ABB RAPID module: P902.mod

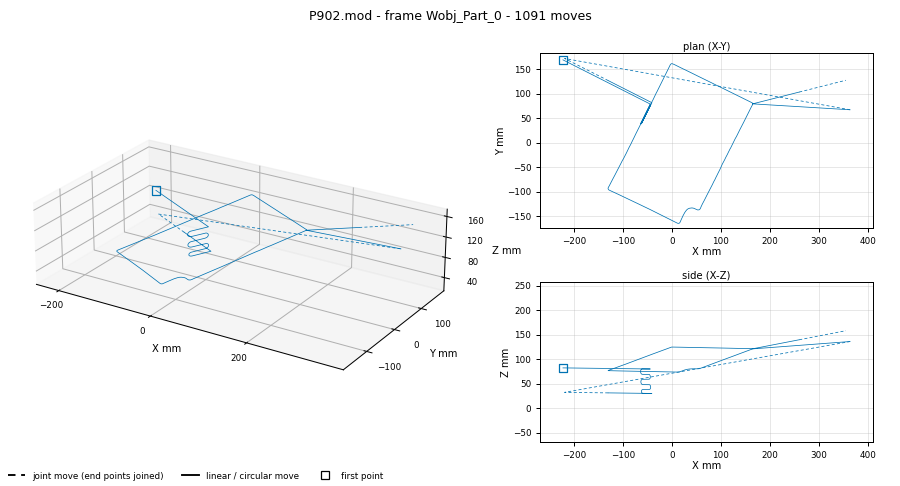
[picture p0: tool path of P902.mod in frame Wobj_Part_0, 1091 of 1101 moves have a stored position in this frame; points joined in program order, loops and branches not executed]
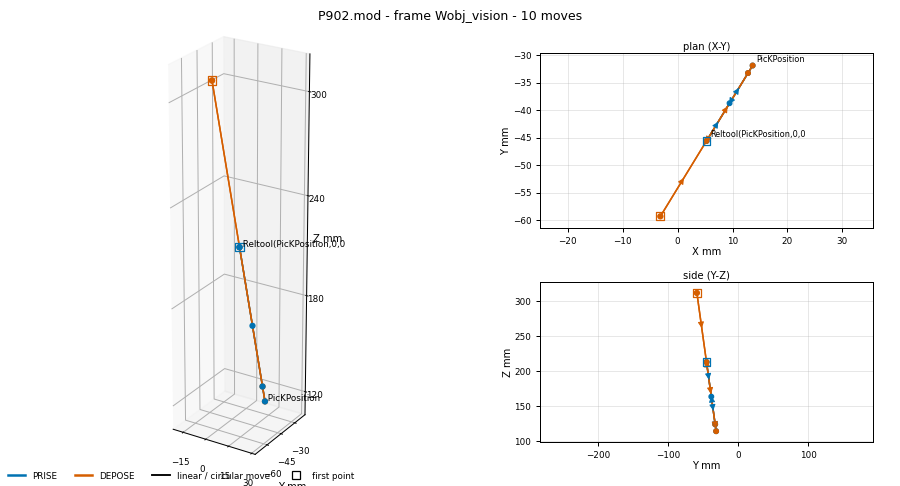
[picture p1: tool path of P902.mod in frame Wobj_vision, 10 of 1101 moves have a stored position in this frame; points joined in program order, loops and branches not executed]
MODULE P902

    ! Nom         :P902
    ! Description :
    ! Créé le     :01/06/2023 14:34:15

    LOCAL CONST SPEEDDATA VitesseLente :=[10,500,0,0];
	LOCAL CONST SPEEDDATA VitesseRapide :=[30,500,0,0];
	LOCAL CONST SPEEDDATA VitesseTronconnage :=[2,500,0,0];
	LOCAL CONST SPEEDDATA VitesseTronconnageApp :=[10,500,0,0];
    !
    !Point de prise
    LOCAL PERS Robtarget PicKPosition := [[13.6622090132406,-31.8672401655374,114.53373902136],[0.0717783424878255,-0.517500201429471,0.851863865981831,0.037004930815311],[0,0,0,0],[8.999999E+09,8.999999E+09,8.999999E+09,8.999999E+09,8.999999E+09,8.999999E+09]];
	LOCAL PERS Pose Ref := [[0,0,0],[1,0,0,0]];
    !
    !Declaration des points de meulage

    !Tr_meulage_motif_1 : Meulage d'un motif
    LOCAL CONST Robtarget Tr_meulage_motif_1_0 := [[-44.4600078125,78.776296875,79.8267421875],[0.368121083594183,-0.372259670766582,0.605815460428718,-0.599080322861418],[0,0,0,0],[8.999999E+09,8.999999E+09,8.999999E+09,8.999999E+09,8.999999E+09,8.999999E+09]];
    LOCAL CONST Robtarget Tr_meulage_motif_1_1 := [[-44.90398828125,77.8802578125,79.82678125],[0.368121083594183,-0.372259670766582,0.605815460428718,-0.599080322861418],[0,0,0,0],[8.999999E+09,8.999999E+09,8.999999E+09,8.999999E+09,8.999999E+09,8.999999E+09]];
    LOCAL CONST Robtarget Tr_meulage_motif_1_2 := [[-45.34796484375,76.98421875,79.8268203125],[0.368121083594183,-0.372259670766582,0.605815460428718,-0.599080322861418],[0,0,0,0],[8.999999E+09,8.999999E+09,8.999999E+09,8.999999E+09,8.999999E+09,8.999999E+09]];
    LOCAL CONST Robtarget Tr_meulage_motif_1_3 := [[-45.7919453125,76.0881796875,79.8268515625],[0.368121083594183,-0.372259670766582,0.605815460428718,-0.599080322861418],[0,0,0,0],[8.999999E+09,8.999999E+09,8.999999E+09,8.999999E+09,8.999999E+09,8.999999E+09]];
    LOCAL CONST Robtarget Tr_meulage_motif_1_4 := [[-46.23592578125,75.1921484375,79.826890625],[0.368121083594183,-0.372259670766582,0.605815460428718,-0.599080322861418],[0,0,0,0],[8.999999E+09,8.999999E+09,8.999999E+09,8.999999E+09,8.999999E+09,8.999999E+09]];
    LOCAL CONST Robtarget Tr_meulage_motif_1_5 := [[-46.67990234375,74.296109375,79.8269296875],[0.368121083594183,-0.372259670766582,0.605815460428718,-0.599080322861418],[0,0,0,0],[8.999999E+09,8.999999E+09,8.999999E+09,8.999999E+09,8.999999E+09,8.999999E+09]];
    LOCAL CONST Robtarget Tr_meulage_motif_1_6 := [[-47.1238828125,73.4000703125,79.82696875],[0.368121083594183,-0.372259670766582,0.605815460428718,-0.599080322861418],[0,0,0,0],[8.999999E+09,8.999999E+09,8.999999E+09,8.999999E+09,8.999999E+09,8.999999E+09]];
    LOCAL CONST Robtarget Tr_meulage_motif_1_7 := [[-47.567859375,72.50403125,79.827],[0.368121083594183,-0.372259670766582,0.605815460428718,-0.599080322861418],[0,0,0,0],[8.999999E+09,8.999999E+09,8.999999E+09,8.999999E+09,8.999999E+09,8.999999E+09]];
    LOCAL CONST Robtarget Tr_meulage_motif_1_8 := [[-48.01183984375,71.608,79.8270390625],[0.368121083594183,-0.372259670766582,0.605815460428718,-0.599080322861418],[0,0,0,0],[8.999999E+09,8.999999E+09,8.999999E+09,8.999999E+09,8.999999E+09,8.999999E+09]];
    LOCAL CONST Robtarget Tr_meulage_motif_1_9 := [[-48.4558203125,70.7119609375,79.827078125],[0.368121083594183,-0.372259670766582,0.605815460428718,-0.599080322861418],[0,0,0,0],[8.999999E+09,8.999999E+09,8.999999E+09,8.999999E+09,8.999999E+09,8.999999E+09]];
    LOCAL CONST Robtarget Tr_meulage_motif_1_10 := [[-48.899796875,69.815921875,79.8271171875],[0.368121083594183,-0.372259670766582,0.605815460428718,-0.599080322861418],[0,0,0,0],[8.999999E+09,8.999999E+09,8.999999E+09,8.999999E+09,8.999999E+09,8.999999E+09]];
    LOCAL CONST Robtarget Tr_meulage_motif_1_11 := [[-49.34377734375,68.9198828125,79.8271484375],[0.368121083594183,-0.372259670766582,0.605815460428718,-0.599080322861418],[0,0,0,0],[8.999999E+09,8.999999E+09,8.999999E+09,8.999999E+09,8.999999E+09,8.999999E+09]];
    LOCAL CONST Robtarget Tr_meulage_motif_1_12 := [[-49.78775390625,68.02384375,79.8271875],[0.368121083594183,-0.372259670766582,0.605815460428718,-0.599080322861418],[0,0,0,0],[8.999999E+09,8.999999E+09,8.999999E+09,8.999999E+09,8.999999E+09,8.999999E+09]];
    LOCAL CONST Robtarget Tr_meulage_motif_1_13 := [[-50.231734375,67.1278125,79.8272265625],[0.368121083594183,-0.372259670766582,0.605815460428718,-0.599080322861418],[0,0,0,0],[8.999999E+09,8.999999E+09,8.999999E+09,8.999999E+09,8.999999E+09,8.999999E+09]];
    LOCAL CONST Robtarget Tr_meulage_motif_1_14 := [[-50.67571484375,66.2317734375,79.827265625],[0.368121083594183,-0.372259670766582,0.605815460428718,-0.599080322861418],[0,0,0,0],[8.999999E+09,8.999999E+09,8.999999E+09,8.999999E+09,8.999999E+09,8.999999E+09]];
    LOCAL CONST Robtarget Tr_meulage_motif_1_15 := [[-51.11969140625,65.335734375,79.827296875],[0.368121083594183,-0.372259670766582,0.605815460428718,-0.599080322861418],[0,0,0,0],[8.999999E+09,8.999999E+09,8.999999E+09,8.999999E+09,8.999999E+09,8.999999E+09]];
    LOCAL CONST Robtarget Tr_meulage_motif_1_16 := [[-51.563671875,64.43969921875,79.8273359375],[0.368121083594183,-0.372259670766582,0.605815460428718,-0.599080322861418],[0,0,0,0],[8.999999E+09,8.999999E+09,8.999999E+09,8.999999E+09,8.999999E+09,8.999999E+09]];
    LOCAL CONST Robtarget Tr_meulage_motif_1_17 := [[-52.00765234375,63.54366015625,79.827375],[0.368121083594183,-0.372259670766582,0.605815460428718,-0.599080322861418],[0,0,0,0],[8.999999E+09,8.999999E+09,8.999999E+09,8.999999E+09,8.999999E+09,8.999999E+09]];
    LOCAL CONST Robtarget Tr_meulage_motif_1_18 := [[-52.45162890625,62.647625,79.8274140625],[0.368121083594183,-0.372259670766582,0.605815460428718,-0.599080322861418],[0,0,0,0],[8.999999E+09,8.999999E+09,8.999999E+09,8.999999E+09,8.999999E+09,8.999999E+09]];
    LOCAL CONST Robtarget Tr_meulage_motif_1_19 := [[-52.895609375,61.7515859375,79.8274453125],[0.368121083594183,-0.372259670766582,0.605815460428718,-0.599080322861418],[0,0,0,0],[8.999999E+09,8.999999E+09,8.999999E+09,8.999999E+09,8.999999E+09,8.999999E+09]];
    LOCAL CONST Robtarget Tr_meulage_motif_1_20 := [[-53.3395859375,60.85555078125,79.827484375],[0.368121083594183,-0.372259670766582,0.605815460428718,-0.599080322861418],[0,0,0,0],[8.999999E+09,8.999999E+09,8.999999E+09,8.999999E+09,8.999999E+09,8.999999E+09]];
    LOCAL CONST Robtarget Tr_meulage_motif_1_21 := [[-53.78356640625,59.95951171875,79.8275234375],[0.368121083594183,-0.372259670766582,0.605815460428718,-0.599080322861418],[0,0,0,0],[8.999999E+09,8.999999E+09,8.999999E+09,8.999999E+09,8.999999E+09,8.999999E+09]];
    LOCAL CONST Robtarget Tr_meulage_motif_1_22 := [[-54.227546875,59.0634765625,79.8275625],[0.368121083594183,-0.372259670766582,0.605815460428718,-0.599080322861418],[0,0,0,0],[8.999999E+09,8.999999E+09,8.999999E+09,8.999999E+09,8.999999E+09,8.999999E+09]];
    LOCAL CONST Robtarget Tr_meulage_motif_1_23 := [[-54.6715234375,58.1674375,79.82759375],[0.368121083594183,-0.372259670766582,0.605815460428718,-0.599080322861418],[0,0,0,0],[8.999999E+09,8.999999E+09,8.999999E+09,8.999999E+09,8.999999E+09,8.999999E+09]];
    LOCAL CONST Robtarget Tr_meulage_motif_1_24 := [[-55.11550390625,57.27140234375,79.8276328125],[0.368121083594183,-0.372259670766582,0.605815460428718,-0.599080322861418],[0,0,0,0],[8.999999E+09,8.999999E+09,8.999999E+09,8.999999E+09,8.999999E+09,8.999999E+09]];
    LOCAL CONST Robtarget Tr_meulage_motif_1_25 := [[-55.55948046875,56.37536328125,79.827671875],[0.368121083594183,-0.372259670766582,0.605815460428718,-0.599080322861418],[0,0,0,0],[8.999999E+09,8.999999E+09,8.999999E+09,8.999999E+09,8.999999E+09,8.999999E+09]];
    LOCAL CONST Robtarget Tr_meulage_motif_1_26 := [[-56.0034609375,55.479328125,79.8277109375],[0.368121083594183,-0.372259670766582,0.605815460428718,-0.599080322861418],[0,0,0,0],[8.999999E+09,8.999999E+09,8.999999E+09,8.999999E+09,8.999999E+09,8.999999E+09]];
    LOCAL CONST Robtarget Tr_meulage_motif_1_27 := [[-56.44744140625,54.5832890625,79.82775],[0.368121083594183,-0.372259670766582,0.605815460428718,-0.599080322861418],[0,0,0,0],[8.999999E+09,8.999999E+09,8.999999E+09,8.999999E+09,8.999999E+09,8.999999E+09]];
    LOCAL CONST Robtarget Tr_meulage_motif_1_28 := [[-56.89141796875,53.68725390625,79.82778125],[0.368121083594183,-0.372259670766582,0.605815460428718,-0.599080322861418],[0,0,0,0],[8.999999E+09,8.999999E+09,8.999999E+09,8.999999E+09,8.999999E+09,8.999999E+09]];
    LOCAL CONST Robtarget Tr_meulage_motif_1_29 := [[-57.3353984375,52.79121484375,79.8278203125],[0.368121083594183,-0.372259670766582,0.605815460428718,-0.599080322861418],[0,0,0,0],[8.999999E+09,8.999999E+09,8.999999E+09,8.999999E+09,8.999999E+09,8.999999E+09]];
    LOCAL CONST Robtarget Tr_meulage_motif_1_30 := [[-57.779375,51.89517578125,79.827859375],[0.368121083594183,-0.372259670766582,0.605815460428718,-0.599080322861418],[0,0,0,0],[8.999999E+09,8.999999E+09,8.999999E+09,8.999999E+09,8.999999E+09,8.999999E+09]];
    LOCAL CONST Robtarget Tr_meulage_motif_1_31 := [[-58.22335546875,50.999140625,79.8278984375],[0.368121083594183,-0.372259670766582,0.605815460428718,-0.599080322861418],[0,0,0,0],[8.999999E+09,8.999999E+09,8.999999E+09,8.999999E+09,8.999999E+09,8.999999E+09]];
    LOCAL CONST Robtarget Tr_meulage_motif_1_32 := [[-58.6673359375,50.1031015625,79.8279296875],[0.368121083594183,-0.372259670766582,0.605815460428718,-0.599080322861418],[0,0,0,0],[8.999999E+09,8.999999E+09,8.999999E+09,8.999999E+09,8.999999E+09,8.999999E+09]];
    LOCAL CONST Robtarget Tr_meulage_motif_1_33 := [[-59.1113125,49.20706640625,79.82796875],[0.368121083594183,-0.372259670766582,0.605815460428718,-0.599080322861418],[0,0,0,0],[8.999999E+09,8.999999E+09,8.999999E+09,8.999999E+09,8.999999E+09,8.999999E+09]];
    LOCAL CONST Robtarget Tr_meulage_motif_1_34 := [[-59.55529296875,48.31102734375,79.8280078125],[0.368121083594183,-0.372259670766582,0.605815460428718,-0.599080322861418],[0,0,0,0],[8.999999E+09,8.999999E+09,8.999999E+09,8.999999E+09,8.999999E+09,8.999999E+09]];
    LOCAL CONST Robtarget Tr_meulage_motif_1_35 := [[-59.99926953125,47.4149921875,79.828046875],[0.368121083594183,-0.372259670766582,0.605815460428718,-0.599080322861418],[0,0,0,0],[8.999999E+09,8.999999E+09,8.999999E+09,8.999999E+09,8.999999E+09,8.999999E+09]];
    LOCAL CONST Robtarget Tr_meulage_motif_1_36 := [[-60.44325,46.518953125,79.828078125],[0.368121083594183,-0.372259670766582,0.605815460428718,-0.599080322861418],[0,0,0,0],[8.999999E+09,8.999999E+09,8.999999E+09,8.999999E+09,8.999999E+09,8.999999E+09]];
    LOCAL CONST Robtarget Tr_meulage_motif_1_37 := [[-60.88723046875,45.62291796875,79.8281171875],[0.368121083594183,-0.372259670766582,0.605815460428718,-0.599080322861418],[0,0,0,0],[8.999999E+09,8.999999E+09,8.999999E+09,8.999999E+09,8.999999E+09,8.999999E+09]];
    LOCAL CONST Robtarget Tr_meulage_motif_1_38 := [[-61.33120703125,44.72687890625,79.82815625],[0.368121083594183,-0.372259670766582,0.605815460428718,-0.599080322861418],[0,0,0,0],[8.999999E+09,8.999999E+09,8.999999E+09,8.999999E+09,8.999999E+09,8.999999E+09]];
    LOCAL CONST Robtarget Tr_meulage_motif_1_39 := [[-61.7684140625,43.83578125,79.7176640625],[0.368121083594183,-0.372259670766582,0.605815460428718,-0.599080322861418],[0,0,0,0],[8.999999E+09,8.999999E+09,8.999999E+09,8.999999E+09,8.999999E+09,8.999999E+09]];
    LOCAL CONST Robtarget Tr_meulage_motif_1_40 := [[-62.182015625,42.984390625,79.506640625],[0.368121083594183,-0.372259670766582,0.605815460428718,-0.599080322861418],[0,0,0,0],[8.999999E+09,8.999999E+09,8.999999E+09,8.999999E+09,8.999999E+09,8.999999E+09]];
    LOCAL CONST Robtarget Tr_meulage_motif_1_41 := [[-62.55207421875,42.2160859375,79.235],[0.368121083594183,-0.372259670766582,0.605815460428718,-0.599080322861418],[0,0,0,0],[8.999999E+09,8.999999E+09,8.999999E+09,8.999999E+09,8.999999E+09,8.999999E+09]];
    LOCAL CONST Robtarget Tr_meulage_motif_1_42 := [[-62.876375,41.5398125,78.9592578125],[0.368121083594183,-0.372259670766582,0.605815460428718,-0.599080322861418],[0,0,0,0],[8.999999E+09,8.999999E+09,8.999999E+09,8.999999E+09,8.999999E+09,8.999999E+09]];
    LOCAL CONST Robtarget Tr_meulage_motif_1_43 := [[-63.34589453125,40.5436171875,78.3435546875],[0.368121083594183,-0.372259670766582,0.605815460428718,-0.599080322861418],[0,0,0,0],[8.999999E+09,8.999999E+09,8.999999E+09,8.999999E+09,8.999999E+09,8.999999E+09]];
    LOCAL CONST Robtarget Tr_meulage_motif_1_44 := [[-63.773875,39.61297265625,77.496453125],[0.368121083594183,-0.372259670766582,0.605815460428718,-0.599080322861418],[0,0,0,0],[8.999999E+09,8.999999E+09,8.999999E+09,8.999999E+09,8.999999E+09,8.999999E+09]];
    LOCAL CONST Robtarget Tr_meulage_motif_1_45 := [[-64.11809375,38.837484375,76.4732421875],[0.368121083594183,-0.372259670766582,0.605815460428718,-0.599080322861418],[0,0,0,0],[8.999999E+09,8.999999E+09,8.999999E+09,8.999999E+09,8.999999E+09,8.999999E+09]];
    LOCAL CONST Robtarget Tr_meulage_motif_1_46 := [[-64.2998046875,38.3826796875,75.3577578125],[0.368121083594183,-0.372259670766582,0.605815460428718,-0.599080322861418],[0,0,0,0],[8.999999E+09,8.999999E+09,8.999999E+09,8.999999E+09,8.999999E+09,8.999999E+09]];
    LOCAL CONST Robtarget Tr_meulage_motif_1_47 := [[-64.289984375,38.34758203125,74.6622109375],[0.368121083594183,-0.372259670766582,0.605815460428718,-0.599080322861418],[0,0,0,0],[8.999999E+09,8.999999E+09,8.999999E+09,8.999999E+09,8.999999E+09,8.999999E+09]];
    LOCAL CONST Robtarget Tr_meulage_motif_1_48 := [[-64.26923828125,38.3372734375,74.0013671875],[0.368121083594183,-0.372259670766582,0.605815460428718,-0.599080322861418],[0,0,0,0],[8.999999E+09,8.999999E+09,8.999999E+09,8.999999E+09,8.999999E+09,8.999999E+09]];
    LOCAL CONST Robtarget Tr_meulage_motif_1_49 := [[-64.2241328125,38.376140625,73.3406796875],[0.368121083594183,-0.372259670766582,0.605815460428718,-0.599080322861418],[0,0,0,0],[8.999999E+09,8.999999E+09,8.999999E+09,8.999999E+09,8.999999E+09,8.999999E+09]];
    LOCAL CONST Robtarget Tr_meulage_motif_1_50 := [[-63.9683671875,38.805390625,72.2395859375],[0.368121083594183,-0.372259670766582,0.605815460428718,-0.599080322861418],[0,0,0,0],[8.999999E+09,8.999999E+09,8.999999E+09,8.999999E+09,8.999999E+09,8.999999E+09]];
    LOCAL CONST Robtarget Tr_meulage_motif_1_51 := [[-63.5564609375,39.557265625,71.233546875],[0.368121083594183,-0.372259670766582,0.605815460428718,-0.599080322861418],[0,0,0,0],[8.999999E+09,8.999999E+09,8.999999E+09,8.999999E+09,8.999999E+09,8.999999E+09]];
    LOCAL CONST Robtarget Tr_meulage_motif_1_52 := [[-63.0760859375,40.46135546875,70.4051484375],[0.368121083594183,-0.372259670766582,0.605815460428718,-0.599080322861418],[0,0,0,0],[8.999999E+09,8.999999E+09,8.999999E+09,8.999999E+09,8.999999E+09,8.999999E+09]];
    LOCAL CONST Robtarget Tr_meulage_motif_1_53 := [[-62.75861328125,41.0708515625,70.009609375],[0.368121083594183,-0.372259670766582,0.605815460428718,-0.599080322861418],[0,0,0,0],[8.999999E+09,8.999999E+09,8.999999E+09,8.999999E+09,8.999999E+09,8.999999E+09]];
    LOCAL CONST Robtarget Tr_meulage_motif_1_54 := [[-62.22912109375,42.101,69.5223359375],[0.368121083594183,-0.372259670766582,0.605815460428718,-0.599080322861418],[0,0,0,0],[8.999999E+09,8.999999E+09,8.999999E+09,8.999999E+09,8.999999E+09,8.999999E+09]];
    LOCAL CONST Robtarget Tr_meulage_motif_1_55 := [[-61.84566015625,42.85406640625,69.258375],[0.368121083594183,-0.372259670766582,0.605815460428718,-0.599080322861418],[0,0,0,0],[8.999999E+09,8.999999E+09,8.999999E+09,8.999999E+09,8.999999E+09,8.999999E+09]];
    LOCAL CONST Robtarget Tr_meulage_motif_1_56 := [[-61.42545703125,43.685984375,69.054],[0.368121083594183,-0.372259670766582,0.605815460428718,-0.599080322861418],[0,0,0,0],[8.999999E+09,8.999999E+09,8.999999E+09,8.999999E+09,8.999999E+09,8.999999E+09]];
    LOCAL CONST Robtarget Tr_meulage_motif_1_57 := [[-60.9862578125,44.56380859375,68.9454296875],[0.368121083594183,-0.372259670766582,0.605815460428718,-0.599080322861418],[0,0,0,0],[8.999999E+09,8.999999E+09,8.999999E+09,8.999999E+09,8.999999E+09,8.999999E+09]];
    LOCAL CONST Robtarget Tr_meulage_motif_1_58 := [[-60.542109375,45.45145703125,68.8348671875],[0.368121083594183,-0.372259670766582,0.605815460428718,-0.599080322861418],[0,0,0,0],[8.999999E+09,8.999999E+09,8.999999E+09,8.999999E+09,8.999999E+09,8.999999E+09]];
    LOCAL CONST Robtarget Tr_meulage_motif_1_59 := [[-60.09812890625,46.34749609375,68.8348359375],[0.368121083594183,-0.372259670766582,0.605815460428718,-0.599080322861418],[0,0,0,0],[8.999999E+09,8.999999E+09,8.999999E+09,8.999999E+09,8.999999E+09,8.999999E+09]];
    LOCAL CONST Robtarget Tr_meulage_motif_1_60 := [[-59.65415234375,47.24353125,68.834796875],[0.368121083594183,-0.372259670766582,0.605815460428718,-0.599080322861418],[0,0,0,0],[8.999999E+09,8.999999E+09,8.999999E+09,8.999999E+09,8.999999E+09,8.999999E+09]];
    LOCAL CONST Robtarget Tr_meulage_motif_1_61 := [[-59.210171875,48.1395703125,68.8347578125],[0.368121083594183,-0.372259670766582,0.605815460428718,-0.599080322861418],[0,0,0,0],[8.999999E+09,8.999999E+09,8.999999E+09,8.999999E+09,8.999999E+09,8.999999E+09]];
    LOCAL CONST Robtarget Tr_meulage_motif_1_62 := [[-58.7661953125,49.03560546875,68.83471875],[0.368121083594183,-0.372259670766582,0.605815460428718,-0.599080322861418],[0,0,0,0],[8.999999E+09,8.999999E+09,8.999999E+09,8.999999E+09,8.999999E+09,8.999999E+09]];
    LOCAL CONST Robtarget Tr_meulage_motif_1_63 := [[-58.32221484375,49.93164453125,68.8346875],[0.368121083594183,-0.372259670766582,0.605815460428718,-0.599080322861418],[0,0,0,0],[8.999999E+09,8.999999E+09,8.999999E+09,8.999999E+09,8.999999E+09,8.999999E+09]];
    LOCAL CONST Robtarget Tr_meulage_motif_1_64 := [[-57.878234375,50.8276796875,68.8346484375],[0.368121083594183,-0.372259670766582,0.605815460428718,-0.599080322861418],[0,0,0,0],[8.999999E+09,8.999999E+09,8.999999E+09,8.999999E+09,8.999999E+09,8.999999E+09]];
    LOCAL CONST Robtarget Tr_meulage_motif_1_65 := [[-57.4342578125,51.72371875,68.834609375],[0.368121083594183,-0.372259670766582,0.605815460428718,-0.599080322861418],[0,0,0,0],[8.999999E+09,8.999999E+09,8.999999E+09,8.999999E+09,8.999999E+09,8.999999E+09]];
    LOCAL CONST Robtarget Tr_meulage_motif_1_66 := [[-56.99027734375,52.61975390625,68.8345703125],[0.368121083594183,-0.372259670766582,0.605815460428718,-0.599080322861418],[0,0,0,0],[8.999999E+09,8.999999E+09,8.999999E+09,8.999999E+09,8.999999E+09,8.999999E+09]];
    LOCAL CONST Robtarget Tr_meulage_motif_1_67 := [[-56.546296875,53.51579296875,68.8345390625],[0.368121083594183,-0.372259670766582,0.605815460428718,-0.599080322861418],[0,0,0,0],[8.999999E+09,8.999999E+09,8.999999E+09,8.999999E+09,8.999999E+09,8.999999E+09]];
    LOCAL CONST Robtarget Tr_meulage_motif_1_68 := [[-56.1023203125,54.411828125,68.8345],[0.368121083594183,-0.372259670766582,0.605815460428718,-0.599080322861418],[0,0,0,0],[8.999999E+09,8.999999E+09,8.999999E+09,8.999999E+09,8.999999E+09,8.999999E+09]];
    LOCAL CONST Robtarget Tr_meulage_motif_1_69 := [[-55.65833984375,55.3078671875,68.8344609375],[0.368121083594183,-0.372259670766582,0.605815460428718,-0.599080322861418],[0,0,0,0],[8.999999E+09,8.999999E+09,8.999999E+09,8.999999E+09,8.999999E+09,8.999999E+09]];
    LOCAL CONST Robtarget Tr_meulage_motif_1_70 := [[-55.21436328125,56.20390234375,68.834421875],[0.368121083594183,-0.372259670766582,0.605815460428718,-0.599080322861418],[0,0,0,0],[8.999999E+09,8.999999E+09,8.999999E+09,8.999999E+09,8.999999E+09,8.999999E+09]];
    LOCAL CONST Robtarget Tr_meulage_motif_1_71 := [[-54.7703828125,57.09994140625,68.834390625],[0.368121083594183,-0.372259670766582,0.605815460428718,-0.599080322861418],[0,0,0,0],[8.999999E+09,8.999999E+09,8.999999E+09,8.999999E+09,8.999999E+09,8.999999E+09]];
    LOCAL CONST Robtarget Tr_meulage_motif_1_72 := [[-54.32640234375,57.9959765625,68.8343515625],[0.368121083594183,-0.372259670766582,0.605815460428718,-0.599080322861418],[0,0,0,0],[8.999999E+09,8.999999E+09,8.999999E+09,8.999999E+09,8.999999E+09,8.999999E+09]];
    LOCAL CONST Robtarget Tr_meulage_motif_1_73 := [[-53.88242578125,58.892015625,68.8343125],[0.368121083594183,-0.372259670766582,0.605815460428718,-0.599080322861418],[0,0,0,0],[8.999999E+09,8.999999E+09,8.999999E+09,8.999999E+09,8.999999E+09,8.999999E+09]];
    LOCAL CONST Robtarget Tr_meulage_motif_1_74 := [[-53.4384453125,59.78805078125,68.8342734375],[0.368121083594183,-0.372259670766582,0.605815460428718,-0.599080322861418],[0,0,0,0],[8.999999E+09,8.999999E+09,8.999999E+09,8.999999E+09,8.999999E+09,8.999999E+09]];
    LOCAL CONST Robtarget Tr_meulage_motif_1_75 := [[-52.99446875,60.68408984375,68.8342421875],[0.368121083594183,-0.372259670766582,0.605815460428718,-0.599080322861418],[0,0,0,0],[8.999999E+09,8.999999E+09,8.999999E+09,8.999999E+09,8.999999E+09,8.999999E+09]];
    LOCAL CONST Robtarget Tr_meulage_motif_1_76 := [[-52.55048828125,61.58012890625,68.834203125],[0.368121083594183,-0.372259670766582,0.605815460428718,-0.599080322861418],[0,0,0,0],[8.999999E+09,8.999999E+09,8.999999E+09,8.999999E+09,8.999999E+09,8.999999E+09]];
    LOCAL CONST Robtarget Tr_meulage_motif_1_77 := [[-52.1065078125,62.4761640625,68.8341640625],[0.368121083594183,-0.372259670766582,0.605815460428718,-0.599080322861418],[0,0,0,0],[8.999999E+09,8.999999E+09,8.999999E+09,8.999999E+09,8.999999E+09,8.999999E+09]];
    LOCAL CONST Robtarget Tr_meulage_motif_1_78 := [[-51.66253125,63.372203125,68.834125],[0.368121083594183,-0.372259670766582,0.605815460428718,-0.599080322861418],[0,0,0,0],[8.999999E+09,8.999999E+09,8.999999E+09,8.999999E+09,8.999999E+09,8.999999E+09]];
    LOCAL CONST Robtarget Tr_meulage_motif_1_79 := [[-51.21855078125,64.26823828125,68.83409375],[0.368121083594183,-0.372259670766582,0.605815460428718,-0.599080322861418],[0,0,0,0],[8.999999E+09,8.999999E+09,8.999999E+09,8.999999E+09,8.999999E+09,8.999999E+09]];
    LOCAL CONST Robtarget Tr_meulage_motif_1_80 := [[-50.77457421875,65.16427734375,68.8340546875],[0.368121083594183,-0.372259670766582,0.605815460428718,-0.599080322861418],[0,0,0,0],[8.999999E+09,8.999999E+09,8.999999E+09,8.999999E+09,8.999999E+09,8.999999E+09]];
    LOCAL CONST Robtarget Tr_meulage_motif_1_81 := [[-50.33059375,66.0603125,68.834015625],[0.368121083594183,-0.372259670766582,0.605815460428718,-0.599080322861418],[0,0,0,0],[8.999999E+09,8.999999E+09,8.999999E+09,8.999999E+09,8.999999E+09,8.999999E+09]];
    LOCAL CONST Robtarget Tr_meulage_motif_1_82 := [[-49.88661328125,66.9563515625,68.8339765625],[0.368121083594183,-0.372259670766582,0.605815460428718,-0.599080322861418],[0,0,0,0],[8.999999E+09,8.999999E+09,8.999999E+09,8.999999E+09,8.999999E+09,8.999999E+09]];
    LOCAL CONST Robtarget Tr_meulage_motif_1_83 := [[-49.44263671875,67.852390625,68.8339375],[0.368121083594183,-0.372259670766582,0.605815460428718,-0.599080322861418],[0,0,0,0],[8.999999E+09,8.999999E+09,8.999999E+09,8.999999E+09,8.999999E+09,8.999999E+09]];
    LOCAL CONST Robtarget Tr_meulage_motif_1_84 := [[-48.99865625,68.748421875,68.83390625],[0.368121083594183,-0.372259670766582,0.605815460428718,-0.599080322861418],[0,0,0,0],[8.999999E+09,8.999999E+09,8.999999E+09,8.999999E+09,8.999999E+09,8.999999E+09]];
    LOCAL CONST Robtarget Tr_meulage_motif_1_85 := [[-48.5546796875,69.6444609375,68.8338671875],[0.368121083594183,-0.372259670766582,0.605815460428718,-0.599080322861418],[0,0,0,0],[8.999999E+09,8.999999E+09,8.999999E+09,8.999999E+09,8.999999E+09,8.999999E+09]];
    LOCAL CONST Robtarget Tr_meulage_motif_1_86 := [[-48.11069921875,70.5405,68.833828125],[0.368121083594183,-0.372259670766582,0.605815460428718,-0.599080322861418],[0,0,0,0],[8.999999E+09,8.999999E+09,8.999999E+09,8.999999E+09,8.999999E+09,8.999999E+09]];
    LOCAL CONST Robtarget Tr_meulage_motif_1_87 := [[-47.66671875,71.4365390625,68.8337890625],[0.368121083594183,-0.372259670766582,0.605815460428718,-0.599080322861418],[0,0,0,0],[8.999999E+09,8.999999E+09,8.999999E+09,8.999999E+09,8.999999E+09,8.999999E+09]];
    LOCAL CONST Robtarget Tr_meulage_motif_1_88 := [[-47.2227421875,72.3325703125,68.8337578125],[0.368121083594183,-0.372259670766582,0.605815460428718,-0.599080322861418],[0,0,0,0],[8.999999E+09,8.999999E+09,8.999999E+09,8.999999E+09,8.999999E+09,8.999999E+09]];
    LOCAL CONST Robtarget Tr_meulage_motif_1_89 := [[-46.77859375,73.2202265625,68.7231953125],[0.368121083594183,-0.372259670766582,0.605815460428718,-0.599080322861418],[0,0,0,0],[8.999999E+09,8.999999E+09,8.999999E+09,8.999999E+09,8.999999E+09,8.999999E+09]];
    LOCAL CONST Robtarget Tr_meulage_motif_1_90 := [[-46.3517421875,74.06503125,68.5121015625],[0.368121083594183,-0.372259670766582,0.605815460428718,-0.599080322861418],[0,0,0,0],[8.999999E+09,8.999999E+09,8.999999E+09,8.999999E+09,8.999999E+09,8.999999E+09]];
    LOCAL CONST Robtarget Tr_meulage_motif_1_91 := [[-45.964625,74.824859375,68.240390625],[0.368121083594183,-0.372259670766582,0.605815460428718,-0.599080322861418],[0,0,0,0],[8.999999E+09,8.999999E+09,8.999999E+09,8.999999E+09,8.999999E+09,8.999999E+09]];
    LOCAL CONST Robtarget Tr_meulage_motif_1_92 := [[-45.63919140625,75.4576484375,67.9363984375],[0.368121083594183,-0.372259670766582,0.605815460428718,-0.599080322861418],[0,0,0,0],[8.999999E+09,8.999999E+09,8.999999E+09,8.999999E+09,8.999999E+09,8.999999E+09]];
    LOCAL CONST Robtarget Tr_meulage_motif_1_93 := [[-45.15912109375,76.3742421875,67.274234375],[0.368121083594183,-0.372259670766582,0.605815460428718,-0.599080322861418],[0,0,0,0],[8.999999E+09,8.999999E+09,8.999999E+09,8.999999E+09,8.999999E+09,8.999999E+09]];
    LOCAL CONST Robtarget Tr_meulage_motif_1_94 := [[-44.7303828125,77.168359375,66.3728125],[0.368121083594183,-0.372259670766582,0.605815460428718,-0.599080322861418],[0,0,0,0],[8.999999E+09,8.999999E+09,8.999999E+09,8.999999E+09,8.999999E+09,8.999999E+09]];
    LOCAL CONST Robtarget Tr_meulage_motif_1_95 := [[-44.460046875,77.63140625,65.32740625],[0.368121083594183,-0.372259670766582,0.605815460428718,-0.599080322861418],[0,0,0,0],[8.999999E+09,8.999999E+09,8.999999E+09,8.999999E+09,8.999999E+09,8.999999E+09]];
    LOCAL CONST Robtarget Tr_meulage_motif_1_96 := [[-44.35626171875,77.786171875,64.63460546875],[0.368121083594183,-0.372259670766582,0.605815460428718,-0.599080322861418],[0,0,0,0],[8.999999E+09,8.999999E+09,8.999999E+09,8.999999E+09,8.999999E+09,8.999999E+09]];
    LOCAL CONST Robtarget Tr_meulage_motif_1_97 := [[-44.3037578125,77.831375,63.86507421875],[0.368121083594183,-0.372259670766582,0.605815460428718,-0.599080322861418],[0,0,0,0],[8.999999E+09,8.999999E+09,8.999999E+09,8.999999E+09,8.999999E+09,8.999999E+09]];
    LOCAL CONST Robtarget Tr_meulage_motif_1_98 := [[-44.3093203125,77.759390625,63.09567578125],[0.368121083594183,-0.372259670766582,0.605815460428718,-0.599080322861418],[0,0,0,0],[8.999999E+09,8.999999E+09,8.999999E+09,8.999999E+09,8.999999E+09,8.999999E+09]];
    LOCAL CONST Robtarget Tr_meulage_motif_1_99 := [[-44.46083984375,77.3661484375,61.98812109375],[0.368121083594183,-0.372259670766582,0.605815460428718,-0.599080322861418],[0,0,0,0],[8.999999E+09,8.999999E+09,8.999999E+09,8.999999E+09,8.999999E+09,8.999999E+09]];
    LOCAL CONST Robtarget Tr_meulage_motif_1_100 := [[-44.62641015625,76.98578125,61.40280859375],[0.368121083594183,-0.372259670766582,0.605815460428718,-0.599080322861418],[0,0,0,0],[8.999999E+09,8.999999E+09,8.999999E+09,8.999999E+09,8.999999E+09,8.999999E+09]];
    LOCAL CONST Robtarget Tr_meulage_motif_1_101 := [[-44.99244140625,76.1770546875,60.51626171875],[0.368121083594183,-0.372259670766582,0.605815460428718,-0.599080322861418],[0,0,0,0],[8.999999E+09,8.999999E+09,8.999999E+09,8.999999E+09,8.999999E+09,8.999999E+09]];
    LOCAL CONST Robtarget Tr_meulage_motif_1_102 := [[-45.2394765625,75.645796875,60.1022265625],[0.368121083594183,-0.372259670766582,0.605815460428718,-0.599080322861418],[0,0,0,0],[8.999999E+09,8.999999E+09,8.999999E+09,8.999999E+09,8.999999E+09,8.999999E+09]];
    LOCAL CONST Robtarget Tr_meulage_motif_1_103 := [[-45.718734375,74.6356328125,59.5585078125],[0.368121083594183,-0.372259670766582,0.605815460428718,-0.599080322861418],[0,0,0,0],[8.999999E+09,8.999999E+09,8.999999E+09,8.999999E+09,8.999999E+09,8.999999E+09]];
    LOCAL CONST Robtarget Tr_meulage_motif_1_104 := [[-46.0760078125,73.891265625,59.26321875],[0.368121083594183,-0.372259670766582,0.605815460428718,-0.599080322861418],[0,0,0,0],[8.999999E+09,8.999999E+09,8.999999E+09,8.999999E+09,8.999999E+09,8.999999E+09]];
    LOCAL CONST Robtarget Tr_meulage_motif_1_105 := [[-46.4833828125,73.05296875,59.05891015625],[0.368121083594183,-0.372259670766582,0.605815460428718,-0.599080322861418],[0,0,0,0],[8.999999E+09,8.999999E+09,8.999999E+09,8.999999E+09,8.999999E+09,8.999999E+09]];
    LOCAL CONST Robtarget Tr_meulage_motif_1_106 := [[-46.915765625,72.1717578125,58.950421875],[0.368121083594183,-0.372259670766582,0.605815460428718,-0.599080322861418],[0,0,0,0],[8.999999E+09,8.999999E+09,8.999999E+09,8.999999E+09,8.999999E+09,8.999999E+09]];
    LOCAL CONST Robtarget Tr_meulage_motif_1_107 := [[-47.35297265625,71.2806640625,58.8399296875],[0.368121083594183,-0.372259670766582,0.605815460428718,-0.599080322861418],[0,0,0,0],[8.999999E+09,8.999999E+09,8.999999E+09,8.999999E+09,8.999999E+09,8.999999E+09]];
    LOCAL CONST Robtarget Tr_meulage_motif_1_108 := [[-47.796953125,70.384625,58.83996875],[0.368121083594183,-0.372259670766582,0.605815460428718,-0.599080322861418],[0,0,0,0],[8.999999E+09,8.999999E+09,8.999999E+09,8.999999E+09,8.999999E+09,8.999999E+09]];
    LOCAL CONST Robtarget Tr_meulage_motif_1_109 := [[-48.24093359375,69.4885859375,58.84000390625],[0.368121083594183,-0.372259670766582,0.605815460428718,-0.599080322861418],[0,0,0,0],[8.999999E+09,8.999999E+09,8.999999E+09,8.999999E+09,8.999999E+09,8.999999E+09]];
    LOCAL CONST Robtarget Tr_meulage_motif_1_110 := [[-48.68491015625,68.5925546875,58.84004296875],[0.368121083594183,-0.372259670766582,0.605815460428718,-0.599080322861418],[0,0,0,0],[8.999999E+09,8.999999E+09,8.999999E+09,8.999999E+09,8.999999E+09,8.999999E+09]];
    LOCAL CONST Robtarget Tr_meulage_motif_1_111 := [[-49.128890625,67.696515625,58.840078125],[0.368121083594183,-0.372259670766582,0.605815460428718,-0.599080322861418],[0,0,0,0],[8.999999E+09,8.999999E+09,8.999999E+09,8.999999E+09,8.999999E+09,8.999999E+09]];
    LOCAL CONST Robtarget Tr_meulage_motif_1_112 := [[-49.57287109375,66.8004765625,58.8401171875],[0.368121083594183,-0.372259670766582,0.605815460428718,-0.599080322861418],[0,0,0,0],[8.999999E+09,8.999999E+09,8.999999E+09,8.999999E+09,8.999999E+09,8.999999E+09]];
    LOCAL CONST Robtarget Tr_meulage_motif_1_113 := [[-50.01684765625,65.9044375,58.84015234375],[0.368121083594183,-0.372259670766582,0.605815460428718,-0.599080322861418],[0,0,0,0],[8.999999E+09,8.999999E+09,8.999999E+09,8.999999E+09,8.999999E+09,8.999999E+09]];
    LOCAL CONST Robtarget Tr_meulage_motif_1_114 := [[-50.460828125,65.00840234375,58.84019140625],[0.368121083594183,-0.372259670766582,0.605815460428718,-0.599080322861418],[0,0,0,0],[8.999999E+09,8.999999E+09,8.999999E+09,8.999999E+09,8.999999E+09,8.999999E+09]];
    LOCAL CONST Robtarget Tr_meulage_motif_1_115 := [[-50.9048046875,64.1123671875,58.8402265625],[0.368121083594183,-0.372259670766582,0.605815460428718,-0.599080322861418],[0,0,0,0],[8.999999E+09,8.999999E+09,8.999999E+09,8.999999E+09,8.999999E+09,8.999999E+09]];
    LOCAL CONST Robtarget Tr_meulage_motif_1_116 := [[-51.34878515625,63.216328125,58.840265625],[0.368121083594183,-0.372259670766582,0.605815460428718,-0.599080322861418],[0,0,0,0],[8.999999E+09,8.999999E+09,8.999999E+09,8.999999E+09,8.999999E+09,8.999999E+09]];
    LOCAL CONST Robtarget Tr_meulage_motif_1_117 := [[-51.792765625,62.32029296875,58.84030078125],[0.368121083594183,-0.372259670766582,0.605815460428718,-0.599080322861418],[0,0,0,0],[8.999999E+09,8.999999E+09,8.999999E+09,8.999999E+09,8.999999E+09,8.999999E+09]];
    LOCAL CONST Robtarget Tr_meulage_motif_1_118 := [[-52.2367421875,61.42425390625,58.84033984375],[0.368121083594183,-0.372259670766582,0.605815460428718,-0.599080322861418],[0,0,0,0],[8.999999E+09,8.999999E+09,8.999999E+09,8.999999E+09,8.999999E+09,8.999999E+09]];
    LOCAL CONST Robtarget Tr_meulage_motif_1_119 := [[-52.68072265625,60.52821875,58.84037890625],[0.368121083594183,-0.372259670766582,0.605815460428718,-0.599080322861418],[0,0,0,0],[8.999999E+09,8.999999E+09,8.999999E+09,8.999999E+09,8.999999E+09,8.999999E+09]];
    LOCAL CONST Robtarget Tr_meulage_motif_1_120 := [[-53.12469921875,59.6321796875,58.8404140625],[0.368121083594183,-0.372259670766582,0.605815460428718,-0.599080322861418],[0,0,0,0],[8.999999E+09,8.999999E+09,8.999999E+09,8.999999E+09,8.999999E+09,8.999999E+09]];
    LOCAL CONST Robtarget Tr_meulage_motif_1_121 := [[-53.5686796875,58.73614453125,58.840453125],[0.368121083594183,-0.372259670766582,0.605815460428718,-0.599080322861418],[0,0,0,0],[8.999999E+09,8.999999E+09,8.999999E+09,8.999999E+09,8.999999E+09,8.999999E+09]];
    LOCAL CONST Robtarget Tr_meulage_motif_1_122 := [[-54.01266015625,57.84010546875,58.84048828125],[0.368121083594183,-0.372259670766582,0.605815460428718,-0.599080322861418],[0,0,0,0],[8.999999E+09,8.999999E+09,8.999999E+09,8.999999E+09,8.999999E+09,8.999999E+09]];
    LOCAL CONST Robtarget Tr_meulage_motif_1_123 := [[-54.45663671875,56.94406640625,58.84052734375],[0.368121083594183,-0.372259670766582,0.605815460428718,-0.599080322861418],[0,0,0,0],[8.999999E+09,8.999999E+09,8.999999E+09,8.999999E+09,8.999999E+09,8.999999E+09]];
    LOCAL CONST Robtarget Tr_meulage_motif_1_124 := [[-54.9006171875,56.04803125,58.8405625],[0.368121083594183,-0.372259670766582,0.605815460428718,-0.599080322861418],[0,0,0,0],[8.999999E+09,8.999999E+09,8.999999E+09,8.999999E+09,8.999999E+09,8.999999E+09]];
    LOCAL CONST Robtarget Tr_meulage_motif_1_125 := [[-55.34459375,55.1519921875,58.8406015625],[0.368121083594183,-0.372259670766582,0.605815460428718,-0.599080322861418],[0,0,0,0],[8.999999E+09,8.999999E+09,8.999999E+09,8.999999E+09,8.999999E+09,8.999999E+09]];
    LOCAL CONST Robtarget Tr_meulage_motif_1_126 := [[-55.78857421875,54.25595703125,58.84063671875],[0.368121083594183,-0.372259670766582,0.605815460428718,-0.599080322861418],[0,0,0,0],[8.999999E+09,8.999999E+09,8.999999E+09,8.999999E+09,8.999999E+09,8.999999E+09]];
    LOCAL CONST Robtarget Tr_meulage_motif_1_127 := [[-56.2325546875,53.35991796875,58.84067578125],[0.368121083594183,-0.372259670766582,0.605815460428718,-0.599080322861418],[0,0,0,0],[8.999999E+09,8.999999E+09,8.999999E+09,8.999999E+09,8.999999E+09,8.999999E+09]];
    LOCAL CONST Robtarget Tr_meulage_motif_1_128 := [[-56.67653125,52.4638828125,58.8407109375],[0.368121083594183,-0.372259670766582,0.605815460428718,-0.599080322861418],[0,0,0,0],[8.999999E+09,8.999999E+09,8.999999E+09,8.999999E+09,8.999999E+09,8.999999E+09]];
    LOCAL CONST Robtarget Tr_meulage_motif_1_129 := [[-57.12051171875,51.56784375,58.84075],[0.368121083594183,-0.372259670766582,0.605815460428718,-0.599080322861418],[0,0,0,0],[8.999999E+09,8.999999E+09,8.999999E+09,8.999999E+09,8.999999E+09,8.999999E+09]];
    LOCAL CONST Robtarget Tr_meulage_motif_1_130 := [[-57.56448828125,50.67180859375,58.84078515625],[0.368121083594183,-0.372259670766582,0.605815460428718,-0.599080322861418],[0,0,0,0],[8.999999E+09,8.999999E+09,8.999999E+09,8.999999E+09,8.999999E+09,8.999999E+09]];
    LOCAL CONST Robtarget Tr_meulage_motif_1_131 := [[-58.00846875,49.77576953125,58.84082421875],[0.368121083594183,-0.372259670766582,0.605815460428718,-0.599080322861418],[0,0,0,0],[8.999999E+09,8.999999E+09,8.999999E+09,8.999999E+09,8.999999E+09,8.999999E+09]];
    LOCAL CONST Robtarget Tr_meulage_motif_1_132 := [[-58.45244921875,48.879734375,58.840859375],[0.368121083594183,-0.372259670766582,0.605815460428718,-0.599080322861418],[0,0,0,0],[8.999999E+09,8.999999E+09,8.999999E+09,8.999999E+09,8.999999E+09,8.999999E+09]];
    LOCAL CONST Robtarget Tr_meulage_motif_1_133 := [[-58.89642578125,47.9836953125,58.8408984375],[0.368121083594183,-0.372259670766582,0.605815460428718,-0.599080322861418],[0,0,0,0],[8.999999E+09,8.999999E+09,8.999999E+09,8.999999E+09,8.999999E+09,8.999999E+09]];
    LOCAL CONST Robtarget Tr_meulage_motif_1_134 := [[-59.34040625,47.08766015625,58.84093359375],[0.368121083594183,-0.372259670766582,0.605815460428718,-0.599080322861418],[0,0,0,0],[8.999999E+09,8.999999E+09,8.999999E+09,8.999999E+09,8.999999E+09,8.999999E+09]];
    LOCAL CONST Robtarget Tr_meulage_motif_1_135 := [[-59.78438671875,46.19162109375,58.84097265625],[0.368121083594183,-0.372259670766582,0.605815460428718,-0.599080322861418],[0,0,0,0],[8.999999E+09,8.999999E+09,8.999999E+09,8.999999E+09,8.999999E+09,8.999999E+09]];
    LOCAL CONST Robtarget Tr_meulage_motif_1_136 := [[-60.22836328125,45.2955859375,58.8410078125],[0.368121083594183,-0.372259670766582,0.605815460428718,-0.599080322861418],[0,0,0,0],[8.999999E+09,8.999999E+09,8.999999E+09,8.999999E+09,8.999999E+09,8.999999E+09]];
    LOCAL CONST Robtarget Tr_meulage_motif_1_137 := [[-60.67234375,44.399546875,58.841046875],[0.368121083594183,-0.372259670766582,0.605815460428718,-0.599080322861418],[0,0,0,0],[8.999999E+09,8.999999E+09,8.999999E+09,8.999999E+09,8.999999E+09,8.999999E+09]];
    LOCAL CONST Robtarget Tr_meulage_motif_1_138 := [[-61.10955078125,43.50844921875,58.73055859375],[0.368121083594183,-0.372259670766582,0.605815460428718,-0.599080322861418],[0,0,0,0],[8.999999E+09,8.999999E+09,8.999999E+09,8.999999E+09,8.999999E+09,8.999999E+09]];
    LOCAL CONST Robtarget Tr_meulage_motif_1_139 := [[-61.5231484375,42.65705859375,58.51953515625],[0.368121083594183,-0.372259670766582,0.605815460428718,-0.599080322861418],[0,0,0,0],[8.999999E+09,8.999999E+09,8.999999E+09,8.999999E+09,8.999999E+09,8.999999E+09]];
    LOCAL CONST Robtarget Tr_meulage_motif_1_140 := [[-61.8932109375,41.88875390625,58.247890625],[0.368121083594183,-0.372259670766582,0.605815460428718,-0.599080322861418],[0,0,0,0],[8.999999E+09,8.999999E+09,8.999999E+09,8.999999E+09,8.999999E+09,8.999999E+09]];
    LOCAL CONST Robtarget Tr_meulage_motif_1_141 := [[-62.2175078125,41.21248046875,57.9721484375],[0.368121083594183,-0.372259670766582,0.605815460428718,-0.599080322861418],[0,0,0,0],[8.999999E+09,8.999999E+09,8.999999E+09,8.999999E+09,8.999999E+09,8.999999E+09]];
    LOCAL CONST Robtarget Tr_meulage_motif_1_142 := [[-62.68702734375,40.21628515625,57.35644140625],[0.368121083594183,-0.372259670766582,0.605815460428718,-0.599080322861418],[0,0,0,0],[8.999999E+09,8.999999E+09,8.999999E+09,8.999999E+09,8.999999E+09,8.999999E+09]];
    LOCAL CONST Robtarget Tr_meulage_motif_1_143 := [[-63.11501171875,39.285640625,56.50934375],[0.368121083594183,-0.372259670766582,0.605815460428718,-0.599080322861418],[0,0,0,0],[8.999999E+09,8.999999E+09,8.999999E+09,8.999999E+09,8.999999E+09,8.999999E+09]];
    LOCAL CONST Robtarget Tr_meulage_motif_1_144 := [[-63.45923046875,38.51015234375,55.48612890625],[0.368121083594183,-0.372259670766582,0.605815460428718,-0.599080322861418],[0,0,0,0],[8.999999E+09,8.999999E+09,8.999999E+09,8.999999E+09,8.999999E+09,8.999999E+09]];
    LOCAL CONST Robtarget Tr_meulage_motif_1_145 := [[-63.64094140625,38.05534765625,54.37064453125],[0.368121083594183,-0.372259670766582,0.605815460428718,-0.599080322861418],[0,0,0,0],[8.999999E+09,8.999999E+09,8.999999E+09,8.999999E+09,8.999999E+09,8.999999E+09]];
    LOCAL CONST Robtarget Tr_meulage_motif_1_146 := [[-63.63112109375,38.02025,53.67510546875],[0.368121083594183,-0.372259670766582,0.605815460428718,-0.599080322861418],[0,0,0,0],[8.999999E+09,8.999999E+09,8.999999E+09,8.999999E+09,8.999999E+09,8.999999E+09]];
    LOCAL CONST Robtarget Tr_meulage_motif_1_147 := [[-63.610375,38.00994140625,53.01426171875],[0.368121083594183,-0.372259670766582,0.605815460428718,-0.599080322861418],[0,0,0,0],[8.999999E+09,8.999999E+09,8.999999E+09,8.999999E+09,8.999999E+09,8.999999E+09]];
    LOCAL CONST Robtarget Tr_meulage_motif_1_148 := [[-63.56526953125,38.04880859375,52.3535703125],[0.368121083594183,-0.372259670766582,0.605815460428718,-0.599080322861418],[0,0,0,0],[8.999999E+09,8.999999E+09,8.999999E+09,8.999999E+09,8.999999E+09,8.999999E+09]];
    LOCAL CONST Robtarget Tr_meulage_motif_1_149 := [[-63.30950390625,38.4780546875,51.25248046875],[0.368121083594183,-0.372259670766582,0.605815460428718,-0.599080322861418],[0,0,0,0],[8.999999E+09,8.999999E+09,8.999999E+09,8.999999E+09,8.999999E+09,8.999999E+09]];
    LOCAL CONST Robtarget Tr_meulage_motif_1_150 := [[-62.89759765625,39.22993359375,50.24644140625],[0.368121083594183,-0.372259670766582,0.605815460428718,-0.599080322861418],[0,0,0,0],[8.999999E+09,8.999999E+09,8.999999E+09,8.999999E+09,8.999999E+09,8.999999E+09]];
    LOCAL CONST Robtarget Tr_meulage_motif_1_151 := [[-62.41721875,40.1340234375,49.41803515625],[0.368121083594183,-0.372259670766582,0.605815460428718,-0.599080322861418],[0,0,0,0],[8.999999E+09,8.999999E+09,8.999999E+09,8.999999E+09,8.999999E+09,8.999999E+09]];
    LOCAL CONST Robtarget Tr_meulage_motif_1_152 := [[-62.09975,40.743515625,49.02250390625],[0.368121083594183,-0.372259670766582,0.605815460428718,-0.599080322861418],[0,0,0,0],[8.999999E+09,8.999999E+09,8.999999E+09,8.999999E+09,8.999999E+09,8.999999E+09]];
    LOCAL CONST Robtarget Tr_meulage_motif_1_153 := [[-61.5702578125,41.77366796875,48.5352265625],[0.368121083594183,-0.372259670766582,0.605815460428718,-0.599080322861418],[0,0,0,0],[8.999999E+09,8.999999E+09,8.999999E+09,8.999999E+09,8.999999E+09,8.999999E+09]];
    LOCAL CONST Robtarget Tr_meulage_motif_1_154 := [[-61.18679296875,42.52673046875,48.271265625],[0.368121083594183,-0.372259670766582,0.605815460428718,-0.599080322861418],[0,0,0,0],[8.999999E+09,8.999999E+09,8.999999E+09,8.999999E+09,8.999999E+09,8.999999E+09]];
    LOCAL CONST Robtarget Tr_meulage_motif_1_155 := [[-60.76658984375,43.35865234375,48.06688671875],[0.368121083594183,-0.372259670766582,0.605815460428718,-0.599080322861418],[0,0,0,0],[8.999999E+09,8.999999E+09,8.999999E+09,8.999999E+09,8.999999E+09,8.999999E+09]];
    LOCAL CONST Robtarget Tr_meulage_motif_1_156 := [[-60.327390625,44.2364765625,47.95832421875],[0.368121083594183,-0.372259670766582,0.605815460428718,-0.599080322861418],[0,0,0,0],[8.999999E+09,8.999999E+09,8.999999E+09,8.999999E+09,8.999999E+09,8.999999E+09]];
    LOCAL CONST Robtarget Tr_meulage_motif_1_157 := [[-59.8832421875,45.124125,47.84776171875],[0.368121083594183,-0.372259670766582,0.605815460428718,-0.599080322861418],[0,0,0,0],[8.999999E+09,8.999999E+09,8.999999E+09,8.999999E+09,8.999999E+09,8.999999E+09]];
    LOCAL CONST Robtarget Tr_meulage_motif_1_158 := [[-59.439265625,46.02016015625,47.84772265625],[0.368121083594183,-0.372259670766582,0.605815460428718,-0.599080322861418],[0,0,0,0],[8.999999E+09,8.999999E+09,8.999999E+09,8.999999E+09,8.999999E+09,8.999999E+09]];
    LOCAL CONST Robtarget Tr_meulage_motif_1_159 := [[-58.99528515625,46.91619921875,47.8476875],[0.368121083594183,-0.372259670766582,0.605815460428718,-0.599080322861418],[0,0,0,0],[8.999999E+09,8.999999E+09,8.999999E+09,8.999999E+09,8.999999E+09,8.999999E+09]];
    LOCAL CONST Robtarget Tr_meulage_motif_1_160 := [[-58.55130859375,47.812234375,47.8476484375],[0.368121083594183,-0.372259670766582,0.605815460428718,-0.599080322861418],[0,0,0,0],[8.999999E+09,8.999999E+09,8.999999E+09,8.999999E+09,8.999999E+09,8.999999E+09]];
    LOCAL CONST Robtarget Tr_meulage_motif_1_161 := [[-58.107328125,48.7082734375,47.84761328125],[0.368121083594183,-0.372259670766582,0.605815460428718,-0.599080322861418],[0,0,0,0],[8.999999E+09,8.999999E+09,8.999999E+09,8.999999E+09,8.999999E+09,8.999999E+09]];
    LOCAL CONST Robtarget Tr_meulage_motif_1_162 := [[-57.66334765625,49.60430859375,47.84757421875],[0.368121083594183,-0.372259670766582,0.605815460428718,-0.599080322861418],[0,0,0,0],[8.999999E+09,8.999999E+09,8.999999E+09,8.999999E+09,8.999999E+09,8.999999E+09]];
    LOCAL CONST Robtarget Tr_meulage_motif_1_163 := [[-57.21937109375,50.50034765625,47.8475390625],[0.368121083594183,-0.372259670766582,0.605815460428718,-0.599080322861418],[0,0,0,0],[8.999999E+09,8.999999E+09,8.999999E+09,8.999999E+09,8.999999E+09,8.999999E+09]];
    LOCAL CONST Robtarget Tr_meulage_motif_1_164 := [[-56.775390625,51.39638671875,47.8475],[0.368121083594183,-0.372259670766582,0.605815460428718,-0.599080322861418],[0,0,0,0],[8.999999E+09,8.999999E+09,8.999999E+09,8.999999E+09,8.999999E+09,8.999999E+09]];
    LOCAL CONST Robtarget Tr_meulage_motif_1_165 := [[-56.3314140625,52.292421875,47.84746484375],[0.368121083594183,-0.372259670766582,0.605815460428718,-0.599080322861418],[0,0,0,0],[8.999999E+09,8.999999E+09,8.999999E+09,8.999999E+09,8.999999E+09,8.999999E+09]];
    LOCAL CONST Robtarget Tr_meulage_motif_1_166 := [[-55.88743359375,53.1884609375,47.84742578125],[0.368121083594183,-0.372259670766582,0.605815460428718,-0.599080322861418],[0,0,0,0],[8.999999E+09,8.999999E+09,8.999999E+09,8.999999E+09,8.999999E+09,8.999999E+09]];
    LOCAL CONST Robtarget Tr_meulage_motif_1_167 := [[-55.443453125,54.08449609375,47.847390625],[0.368121083594183,-0.372259670766582,0.605815460428718,-0.599080322861418],[0,0,0,0],[8.999999E+09,8.999999E+09,8.999999E+09,8.999999E+09,8.999999E+09,8.999999E+09]];
    LOCAL CONST Robtarget Tr_meulage_motif_1_168 := [[-54.9994765625,54.98053515625,47.8473515625],[0.368121083594183,-0.372259670766582,0.605815460428718,-0.599080322861418],[0,0,0,0],[8.999999E+09,8.999999E+09,8.999999E+09,8.999999E+09,8.999999E+09,8.999999E+09]];
    LOCAL CONST Robtarget Tr_meulage_motif_1_169 := [[-54.55549609375,55.8765703125,47.84731640625],[0.368121083594183,-0.372259670766582,0.605815460428718,-0.599080322861418],[0,0,0,0],[8.999999E+09,8.999999E+09,8.999999E+09,8.999999E+09,8.999999E+09,8.999999E+09]];
    LOCAL CONST Robtarget Tr_meulage_motif_1_170 := [[-54.111515625,56.772609375,47.84727734375],[0.368121083594183,-0.372259670766582,0.605815460428718,-0.599080322861418],[0,0,0,0],[8.999999E+09,8.999999E+09,8.999999E+09,8.999999E+09,8.999999E+09,8.999999E+09]];
    LOCAL CONST Robtarget Tr_meulage_motif_1_171 := [[-53.6675390625,57.66864453125,47.8472421875],[0.368121083594183,-0.372259670766582,0.605815460428718,-0.599080322861418],[0,0,0,0],[8.999999E+09,8.999999E+09,8.999999E+09,8.999999E+09,8.999999E+09,8.999999E+09]];
    LOCAL CONST Robtarget Tr_meulage_motif_1_172 := [[-53.22355859375,58.56468359375,47.847203125],[0.368121083594183,-0.372259670766582,0.605815460428718,-0.599080322861418],[0,0,0,0],[8.999999E+09,8.999999E+09,8.999999E+09,8.999999E+09,8.999999E+09,8.999999E+09]];
    LOCAL CONST Robtarget Tr_meulage_motif_1_173 := [[-52.77958203125,59.46071875,47.84716796875],[0.368121083594183,-0.372259670766582,0.605815460428718,-0.599080322861418],[0,0,0,0],[8.999999E+09,8.999999E+09,8.999999E+09,8.999999E+09,8.999999E+09,8.999999E+09]];
    LOCAL CONST Robtarget Tr_meulage_motif_1_174 := [[-52.3356015625,60.3567578125,47.84712890625],[0.368121083594183,-0.372259670766582,0.605815460428718,-0.599080322861418],[0,0,0,0],[8.999999E+09,8.999999E+09,8.999999E+09,8.999999E+09,8.999999E+09,8.999999E+09]];
    LOCAL CONST Robtarget Tr_meulage_motif_1_175 := [[-51.89162109375,61.25279296875,47.84709375],[0.368121083594183,-0.372259670766582,0.605815460428718,-0.599080322861418],[0,0,0,0],[8.999999E+09,8.999999E+09,8.999999E+09,8.999999E+09,8.999999E+09,8.999999E+09]];
    LOCAL CONST Robtarget Tr_meulage_motif_1_176 := [[-51.44764453125,62.14883203125,47.8470546875],[0.368121083594183,-0.372259670766582,0.605815460428718,-0.599080322861418],[0,0,0,0],[8.999999E+09,8.999999E+09,8.999999E+09,8.999999E+09,8.999999E+09,8.999999E+09]];
    LOCAL CONST Robtarget Tr_meulage_motif_1_177 := [[-51.0036640625,63.0448671875,47.84701953125],[0.368121083594183,-0.372259670766582,0.605815460428718,-0.599080322861418],[0,0,0,0],[8.999999E+09,8.999999E+09,8.999999E+09,8.999999E+09,8.999999E+09,8.999999E+09]];
    LOCAL CONST Robtarget Tr_meulage_motif_1_178 := [[-50.5596875,63.94090625,47.84698046875],[0.368121083594183,-0.372259670766582,0.605815460428718,-0.599080322861418],[0,0,0,0],[8.999999E+09,8.999999E+09,8.999999E+09,8.999999E+09,8.999999E+09,8.999999E+09]];
    LOCAL CONST Robtarget Tr_meulage_motif_1_179 := [[-50.11570703125,64.83694140625,47.8469453125],[0.368121083594183,-0.372259670766582,0.605815460428718,-0.599080322861418],[0,0,0,0],[8.999999E+09,8.999999E+09,8.999999E+09,8.999999E+09,8.999999E+09,8.999999E+09]];
    LOCAL CONST Robtarget Tr_meulage_motif_1_180 := [[-49.6717265625,65.7329765625,47.84690625],[0.368121083594183,-0.372259670766582,0.605815460428718,-0.599080322861418],[0,0,0,0],[8.999999E+09,8.999999E+09,8.999999E+09,8.999999E+09,8.999999E+09,8.999999E+09]];
    LOCAL CONST Robtarget Tr_meulage_motif_1_181 := [[-49.22775,66.629015625,47.84687109375],[0.368121083594183,-0.372259670766582,0.605815460428718,-0.599080322861418],[0,0,0,0],[8.999999E+09,8.999999E+09,8.999999E+09,8.999999E+09,8.999999E+09,8.999999E+09]];
    LOCAL CONST Robtarget Tr_meulage_motif_1_182 := [[-48.78376953125,67.5250546875,47.84683203125],[0.368121083594183,-0.372259670766582,0.605815460428718,-0.599080322861418],[0,0,0,0],[8.999999E+09,8.999999E+09,8.999999E+09,8.999999E+09,8.999999E+09,8.999999E+09]];
    LOCAL CONST Robtarget Tr_meulage_motif_1_183 := [[-48.33979296875,68.42109375,47.846796875],[0.368121083594183,-0.372259670766582,0.605815460428718,-0.599080322861418],[0,0,0,0],[8.999999E+09,8.999999E+09,8.999999E+09,8.999999E+09,8.999999E+09,8.999999E+09]];
    LOCAL CONST Robtarget Tr_meulage_motif_1_184 := [[-47.8958125,69.3171328125,47.8467578125],[0.368121083594183,-0.372259670766582,0.605815460428718,-0.599080322861418],[0,0,0,0],[8.999999E+09,8.999999E+09,8.999999E+09,8.999999E+09,8.999999E+09,8.999999E+09]];
    LOCAL CONST Robtarget Tr_meulage_motif_1_185 := [[-47.45183203125,70.2131640625,47.84671875],[0.368121083594183,-0.372259670766582,0.605815460428718,-0.599080322861418],[0,0,0,0],[8.999999E+09,8.999999E+09,8.999999E+09,8.999999E+09,8.999999E+09,8.999999E+09]];
    LOCAL CONST Robtarget Tr_meulage_motif_1_186 := [[-47.00785546875,71.109203125,47.84668359375],[0.368121083594183,-0.372259670766582,0.605815460428718,-0.599080322861418],[0,0,0,0],[8.999999E+09,8.999999E+09,8.999999E+09,8.999999E+09,8.999999E+09,8.999999E+09]];
    LOCAL CONST Robtarget Tr_meulage_motif_1_187 := [[-46.563875,72.0052421875,47.84664453125],[0.368121083594183,-0.372259670766582,0.605815460428718,-0.599080322861418],[0,0,0,0],[8.999999E+09,8.999999E+09,8.999999E+09,8.999999E+09,8.999999E+09,8.999999E+09]];
    LOCAL CONST Robtarget Tr_meulage_motif_1_188 := [[-46.11973046875,72.892890625,47.73608203125],[0.368121083594183,-0.372259670766582,0.605815460428718,-0.599080322861418],[0,0,0,0],[8.999999E+09,8.999999E+09,8.999999E+09,8.999999E+09,8.999999E+09,8.999999E+09]];
    LOCAL CONST Robtarget Tr_meulage_motif_1_189 := [[-45.692875,73.7376953125,47.5249921875],[0.368121083594183,-0.372259670766582,0.605815460428718,-0.599080322861418],[0,0,0,0],[8.999999E+09,8.999999E+09,8.999999E+09,8.999999E+09,8.999999E+09,8.999999E+09]];
    LOCAL CONST Robtarget Tr_meulage_motif_1_190 := [[-45.3057578125,74.49753125,47.25328125],[0.368121083594183,-0.372259670766582,0.605815460428718,-0.599080322861418],[0,0,0,0],[8.999999E+09,8.999999E+09,8.999999E+09,8.999999E+09,8.999999E+09,8.999999E+09]];
    LOCAL CONST Robtarget Tr_meulage_motif_1_191 := [[-44.98032421875,75.1303203125,46.94930078125],[0.368121083594183,-0.372259670766582,0.605815460428718,-0.599080322861418],[0,0,0,0],[8.999999E+09,8.999999E+09,8.999999E+09,8.999999E+09,8.999999E+09,8.999999E+09]];
    LOCAL CONST Robtarget Tr_meulage_motif_1_192 := [[-44.5002578125,76.0469140625,46.28713671875],[0.368121083594183,-0.372259670766582,0.605815460428718,-0.599080322861418],[0,0,0,0],[8.999999E+09,8.999999E+09,8.999999E+09,8.999999E+09,8.999999E+09,8.999999E+09]];
    LOCAL CONST Robtarget Tr_meulage_motif_1_193 := [[-44.071515625,76.8410234375,45.38570703125],[0.368121083594183,-0.372259670766582,0.605815460428718,-0.599080322861418],[0,0,0,0],[8.999999E+09,8.999999E+09,8.999999E+09,8.999999E+09,8.999999E+09,8.999999E+09]];
    LOCAL CONST Robtarget Tr_meulage_motif_1_194 := [[-43.80118359375,77.3040703125,44.3403125],[0.368121083594183,-0.372259670766582,0.605815460428718,-0.599080322861418],[0,0,0,0],[8.999999E+09,8.999999E+09,8.999999E+09,8.999999E+09,8.999999E+09,8.999999E+09]];
    LOCAL CONST Robtarget Tr_meulage_motif_1_195 := [[-43.69739453125,77.4588359375,43.64749609375],[0.368121083594183,-0.372259670766582,0.605815460428718,-0.599080322861418],[0,0,0,0],[8.999999E+09,8.999999E+09,8.999999E+09,8.999999E+09,8.999999E+09,8.999999E+09]];
    LOCAL CONST Robtarget Tr_meulage_motif_1_196 := [[-43.644890625,77.5040390625,42.87796875],[0.368121083594183,-0.372259670766582,0.605815460428718,-0.599080322861418],[0,0,0,0],[8.999999E+09,8.999999E+09,8.999999E+09,8.999999E+09,8.999999E+09,8.999999E+09]];
    LOCAL CONST Robtarget Tr_meulage_motif_1_197 := [[-43.65045703125,77.4320625,42.10858203125],[0.368121083594183,-0.372259670766582,0.605815460428718,-0.599080322861418],[0,0,0,0],[8.999999E+09,8.999999E+09,8.999999E+09,8.999999E+09,8.999999E+09,8.999999E+09]];
    LOCAL CONST Robtarget Tr_meulage_motif_1_198 := [[-43.8019765625,77.0388125,41.00102734375],[0.368121083594183,-0.372259670766582,0.605815460428718,-0.599080322861418],[0,0,0,0],[8.999999E+09,8.999999E+09,8.999999E+09,8.999999E+09,8.999999E+09,8.999999E+09]];
    LOCAL CONST Robtarget Tr_meulage_motif_1_199 := [[-43.967546875,76.6584453125,40.41571484375],[0.368121083594183,-0.372259670766582,0.605815460428718,-0.599080322861418],[0,0,0,0],[8.999999E+09,8.999999E+09,8.999999E+09,8.999999E+09,8.999999E+09,8.999999E+09]];
    LOCAL CONST Robtarget Tr_meulage_motif_1_200 := [[-44.333578125,75.84971875,39.52913671875],[0.368121083594183,-0.372259670766582,0.605815460428718,-0.599080322861418],[0,0,0,0],[8.999999E+09,8.999999E+09,8.999999E+09,8.999999E+09,8.999999E+09,8.999999E+09]];
    LOCAL CONST Robtarget Tr_meulage_motif_1_201 := [[-44.58061328125,75.31846875,39.1151328125],[0.368121083594183,-0.372259670766582,0.605815460428718,-0.599080322861418],[0,0,0,0],[8.999999E+09,8.999999E+09,8.999999E+09,8.999999E+09,8.999999E+09,8.999999E+09]];
    LOCAL CONST Robtarget Tr_meulage_motif_1_202 := [[-45.0598671875,74.308296875,38.5713828125],[0.368121083594183,-0.372259670766582,0.605815460428718,-0.599080322861418],[0,0,0,0],[8.999999E+09,8.999999E+09,8.999999E+09,8.999999E+09,8.999999E+09,8.999999E+09]];
    LOCAL CONST Robtarget Tr_meulage_motif_1_203 := [[-45.417140625,73.5639296875,38.27609375],[0.368121083594183,-0.372259670766582,0.605815460428718,-0.599080322861418],[0,0,0,0],[8.999999E+09,8.999999E+09,8.999999E+09,8.999999E+09,8.999999E+09,8.999999E+09]];
    LOCAL CONST Robtarget Tr_meulage_motif_1_204 := [[-45.824515625,72.7256328125,38.07176953125],[0.368121083594183,-0.372259670766582,0.605815460428718,-0.599080322861418],[0,0,0,0],[8.999999E+09,8.999999E+09,8.999999E+09,8.999999E+09,8.999999E+09,8.999999E+09]];
    LOCAL CONST Robtarget Tr_meulage_motif_1_205 := [[-46.25690234375,71.8444296875,37.963328125],[0.368121083594183,-0.372259670766582,0.605815460428718,-0.599080322861418],[0,0,0,0],[8.999999E+09,8.999999E+09,8.999999E+09,8.999999E+09,8.999999E+09,8.999999E+09]];
    LOCAL CONST Robtarget Tr_meulage_motif_1_206 := [[-46.694109375,70.953328125,37.8528203125],[0.368121083594183,-0.372259670766582,0.605815460428718,-0.599080322861418],[0,0,0,0],[8.999999E+09,8.999999E+09,8.999999E+09,8.999999E+09,8.999999E+09,8.999999E+09]];
    LOCAL CONST Robtarget Tr_meulage_motif_1_207 := [[-47.1380859375,70.057296875,37.852859375],[0.368121083594183,-0.372259670766582,0.605815460428718,-0.599080322861418],[0,0,0,0],[8.999999E+09,8.999999E+09,8.999999E+09,8.999999E+09,8.999999E+09,8.999999E+09]];
    LOCAL CONST Robtarget Tr_meulage_motif_1_208 := [[-47.58206640625,69.1612578125,37.85289453125],[0.368121083594183,-0.372259670766582,0.605815460428718,-0.599080322861418],[0,0,0,0],[8.999999E+09,8.999999E+09,8.999999E+09,8.999999E+09,8.999999E+09,8.999999E+09]];
    LOCAL CONST Robtarget Tr_meulage_motif_1_209 := [[-48.026046875,68.26521875,37.85293359375],[0.368121083594183,-0.372259670766582,0.605815460428718,-0.599080322861418],[0,0,0,0],[8.999999E+09,8.999999E+09,8.999999E+09,8.999999E+09,8.999999E+09,8.999999E+09]];
    LOCAL CONST Robtarget Tr_meulage_motif_1_210 := [[-48.4700234375,67.3691796875,37.85296875],[0.368121083594183,-0.372259670766582,0.605815460428718,-0.599080322861418],[0,0,0,0],[8.999999E+09,8.999999E+09,8.999999E+09,8.999999E+09,8.999999E+09,8.999999E+09]];
    LOCAL CONST Robtarget Tr_meulage_motif_1_211 := [[-48.91400390625,66.4731484375,37.8530078125],[0.368121083594183,-0.372259670766582,0.605815460428718,-0.599080322861418],[0,0,0,0],[8.999999E+09,8.999999E+09,8.999999E+09,8.999999E+09,8.999999E+09,8.999999E+09]];
    LOCAL CONST Robtarget Tr_meulage_motif_1_212 := [[-49.357984375,65.577109375,37.853046875],[0.368121083594183,-0.372259670766582,0.605815460428718,-0.599080322861418],[0,0,0,0],[8.999999E+09,8.999999E+09,8.999999E+09,8.999999E+09,8.999999E+09,8.999999E+09]];
    LOCAL CONST Robtarget Tr_meulage_motif_1_213 := [[-49.8019609375,64.6810703125,37.85308203125],[0.368121083594183,-0.372259670766582,0.605815460428718,-0.599080322861418],[0,0,0,0],[8.999999E+09,8.999999E+09,8.999999E+09,8.999999E+09,8.999999E+09,8.999999E+09]];
    LOCAL CONST Robtarget Tr_meulage_motif_1_214 := [[-50.24594140625,63.78503515625,37.85312109375],[0.368121083594183,-0.372259670766582,0.605815460428718,-0.599080322861418],[0,0,0,0],[8.999999E+09,8.999999E+09,8.999999E+09,8.999999E+09,8.999999E+09,8.999999E+09]];
    LOCAL CONST Robtarget Tr_meulage_motif_1_215 := [[-50.68991796875,62.88899609375,37.85315625],[0.368121083594183,-0.372259670766582,0.605815460428718,-0.599080322861418],[0,0,0,0],[8.999999E+09,8.999999E+09,8.999999E+09,8.999999E+09,8.999999E+09,8.999999E+09]];
    LOCAL CONST Robtarget Tr_meulage_motif_1_216 := [[-51.1338984375,61.99295703125,37.8531953125],[0.368121083594183,-0.372259670766582,0.605815460428718,-0.599080322861418],[0,0,0,0],[8.999999E+09,8.999999E+09,8.999999E+09,8.999999E+09,8.999999E+09,8.999999E+09]];
    LOCAL CONST Robtarget Tr_meulage_motif_1_217 := [[-51.57787890625,61.096921875,37.85323046875],[0.368121083594183,-0.372259670766582,0.605815460428718,-0.599080322861418],[0,0,0,0],[8.999999E+09,8.999999E+09,8.999999E+09,8.999999E+09,8.999999E+09,8.999999E+09]];
    LOCAL CONST Robtarget Tr_meulage_motif_1_218 := [[-52.02185546875,60.2008828125,37.85326953125],[0.368121083594183,-0.372259670766582,0.605815460428718,-0.599080322861418],[0,0,0,0],[8.999999E+09,8.999999E+09,8.999999E+09,8.999999E+09,8.999999E+09,8.999999E+09]];
    LOCAL CONST Robtarget Tr_meulage_motif_1_219 := [[-52.4658359375,59.30484765625,37.8533046875],[0.368121083594183,-0.372259670766582,0.605815460428718,-0.599080322861418],[0,0,0,0],[8.999999E+09,8.999999E+09,8.999999E+09,8.999999E+09,8.999999E+09,8.999999E+09]];
    LOCAL CONST Robtarget Tr_meulage_motif_1_220 := [[-52.9098125,58.40880859375,37.85334375],[0.368121083594183,-0.372259670766582,0.605815460428718,-0.599080322861418],[0,0,0,0],[8.999999E+09,8.999999E+09,8.999999E+09,8.999999E+09,8.999999E+09,8.999999E+09]];
    LOCAL CONST Robtarget Tr_meulage_motif_1_221 := [[-53.35379296875,57.5127734375,37.85337890625],[0.368121083594183,-0.372259670766582,0.605815460428718,-0.599080322861418],[0,0,0,0],[8.999999E+09,8.999999E+09,8.999999E+09,8.999999E+09,8.999999E+09,8.999999E+09]];
    LOCAL CONST Robtarget Tr_meulage_motif_1_222 := [[-53.7977734375,56.616734375,37.85341796875],[0.368121083594183,-0.372259670766582,0.605815460428718,-0.599080322861418],[0,0,0,0],[8.999999E+09,8.999999E+09,8.999999E+09,8.999999E+09,8.999999E+09,8.999999E+09]];
    LOCAL CONST Robtarget Tr_meulage_motif_1_223 := [[-54.24175,55.72069921875,37.853453125],[0.368121083594183,-0.372259670766582,0.605815460428718,-0.599080322861418],[0,0,0,0],[8.999999E+09,8.999999E+09,8.999999E+09,8.999999E+09,8.999999E+09,8.999999E+09]];
    LOCAL CONST Robtarget Tr_meulage_motif_1_224 := [[-54.68573046875,54.82466015625,37.8534921875],[0.368121083594183,-0.372259670766582,0.605815460428718,-0.599080322861418],[0,0,0,0],[8.999999E+09,8.999999E+09,8.999999E+09,8.999999E+09,8.999999E+09,8.999999E+09]];
    LOCAL CONST Robtarget Tr_meulage_motif_1_225 := [[-55.12970703125,53.928625,37.85352734375],[0.368121083594183,-0.372259670766582,0.605815460428718,-0.599080322861418],[0,0,0,0],[8.999999E+09,8.999999E+09,8.999999E+09,8.999999E+09,8.999999E+09,8.999999E+09]];
    LOCAL CONST Robtarget Tr_meulage_motif_1_226 := [[-55.5736875,53.0325859375,37.85356640625],[0.368121083594183,-0.372259670766582,0.605815460428718,-0.599080322861418],[0,0,0,0],[8.999999E+09,8.999999E+09,8.999999E+09,8.999999E+09,8.999999E+09,8.999999E+09]];
    LOCAL CONST Robtarget Tr_meulage_motif_1_227 := [[-56.01766796875,52.13655078125,37.8536015625],[0.368121083594183,-0.372259670766582,0.605815460428718,-0.599080322861418],[0,0,0,0],[8.999999E+09,8.999999E+09,8.999999E+09,8.999999E+09,8.999999E+09,8.999999E+09]];
    LOCAL CONST Robtarget Tr_meulage_motif_1_228 := [[-56.46164453125,51.24051171875,37.853640625],[0.368121083594183,-0.372259670766582,0.605815460428718,-0.599080322861418],[0,0,0,0],[8.999999E+09,8.999999E+09,8.999999E+09,8.999999E+09,8.999999E+09,8.999999E+09]];
    LOCAL CONST Robtarget Tr_meulage_motif_1_229 := [[-56.905625,50.3444765625,37.85367578125],[0.368121083594183,-0.372259670766582,0.605815460428718,-0.599080322861418],[0,0,0,0],[8.999999E+09,8.999999E+09,8.999999E+09,8.999999E+09,8.999999E+09,8.999999E+09]];
    LOCAL CONST Robtarget Tr_meulage_motif_1_230 := [[-57.3496015625,49.4484375,37.85371484375],[0.368121083594183,-0.372259670766582,0.605815460428718,-0.599080322861418],[0,0,0,0],[8.999999E+09,8.999999E+09,8.999999E+09,8.999999E+09,8.999999E+09,8.999999E+09]];
    LOCAL CONST Robtarget Tr_meulage_motif_1_231 := [[-57.79358203125,48.55240234375,37.85375],[0.368121083594183,-0.372259670766582,0.605815460428718,-0.599080322861418],[0,0,0,0],[8.999999E+09,8.999999E+09,8.999999E+09,8.999999E+09,8.999999E+09,8.999999E+09]];
    LOCAL CONST Robtarget Tr_meulage_motif_1_232 := [[-58.2375625,47.65636328125,37.8537890625],[0.368121083594183,-0.372259670766582,0.605815460428718,-0.599080322861418],[0,0,0,0],[8.999999E+09,8.999999E+09,8.999999E+09,8.999999E+09,8.999999E+09,8.999999E+09]];
    LOCAL CONST Robtarget Tr_meulage_motif_1_233 := [[-58.6815390625,46.76032421875,37.85382421875],[0.368121083594183,-0.372259670766582,0.605815460428718,-0.599080322861418],[0,0,0,0],[8.999999E+09,8.999999E+09,8.999999E+09,8.999999E+09,8.999999E+09,8.999999E+09]];
    LOCAL CONST Robtarget Tr_meulage_motif_1_234 := [[-59.12551953125,45.8642890625,37.85386328125],[0.368121083594183,-0.372259670766582,0.605815460428718,-0.599080322861418],[0,0,0,0],[8.999999E+09,8.999999E+09,8.999999E+09,8.999999E+09,8.999999E+09,8.999999E+09]];
    LOCAL CONST Robtarget Tr_meulage_motif_1_235 := [[-59.5695,44.96825,37.8538984375],[0.368121083594183,-0.372259670766582,0.605815460428718,-0.599080322861418],[0,0,0,0],[8.999999E+09,8.999999E+09,8.999999E+09,8.999999E+09,8.999999E+09,8.999999E+09]];
    LOCAL CONST Robtarget Tr_meulage_motif_1_236 := [[-60.0134765625,44.07221484375,37.8539375],[0.368121083594183,-0.372259670766582,0.605815460428718,-0.599080322861418],[0,0,0,0],[8.999999E+09,8.999999E+09,8.999999E+09,8.999999E+09,8.999999E+09,8.999999E+09]];
    LOCAL CONST Robtarget Tr_meulage_motif_1_237 := [[-60.45068359375,43.1811171875,37.74343359375],[0.368121083594183,-0.372259670766582,0.605815460428718,-0.599080322861418],[0,0,0,0],[8.999999E+09,8.999999E+09,8.999999E+09,8.999999E+09,8.999999E+09,8.999999E+09]];
    LOCAL CONST Robtarget Tr_meulage_motif_1_238 := [[-60.86428515625,42.3297265625,37.53241015625],[0.368121083594183,-0.372259670766582,0.605815460428718,-0.599080322861418],[0,0,0,0],[8.999999E+09,8.999999E+09,8.999999E+09,8.999999E+09,8.999999E+09,8.999999E+09]];
    LOCAL CONST Robtarget Tr_meulage_motif_1_239 := [[-61.23434375,41.561421875,37.26078125],[0.368121083594183,-0.372259670766582,0.605815460428718,-0.599080322861418],[0,0,0,0],[8.999999E+09,8.999999E+09,8.999999E+09,8.999999E+09,8.999999E+09,8.999999E+09]];
    LOCAL CONST Robtarget Tr_meulage_motif_1_240 := [[-61.54069140625,40.9191484375,36.9568515625],[0.368121083594183,-0.372259670766582,0.605815460428718,-0.599080322861418],[0,0,0,0],[8.999999E+09,8.999999E+09,8.999999E+09,8.999999E+09,8.999999E+09,8.999999E+09]];
    LOCAL CONST Robtarget Tr_meulage_motif_1_241 := [[-61.9791875,39.98190234375,36.294765625],[0.368121083594183,-0.372259670766582,0.605815460428718,-0.599080322861418],[0,0,0,0],[8.999999E+09,8.999999E+09,8.999999E+09,8.999999E+09,8.999999E+09,8.999999E+09]];
    LOCAL CONST Robtarget Tr_meulage_motif_1_242 := [[-62.3106015625,39.23888671875,35.35559375],[0.368121083594183,-0.372259670766582,0.605815460428718,-0.599080322861418],[0,0,0,0],[8.999999E+09,8.999999E+09,8.999999E+09,8.999999E+09,8.999999E+09,8.999999E+09]];
    LOCAL CONST Robtarget Tr_meulage_motif_1_243 := [[-62.43581640625,38.90755859375,34.35985546875],[0.368121083594183,-0.372259670766582,0.605815460428718,-0.599080322861418],[0,0,0,0],[8.999999E+09,8.999999E+09,8.999999E+09,8.999999E+09,8.999999E+09,8.999999E+09]];
    LOCAL CONST Robtarget Tr_meulage_motif_1_244 := [[-62.40515625,38.92544140625,33.80265234375],[0.368121083594183,-0.372259670766582,0.605815460428718,-0.599080322861418],[0,0,0,0],[8.999999E+09,8.999999E+09,8.999999E+09,8.999999E+09,8.999999E+09,8.999999E+09]];
    LOCAL CONST Robtarget Tr_meulage_motif_1_245 := [[-62.3939609375,38.9150625,33.38500390625],[0.368121083594183,-0.372259670766582,0.605815460428718,-0.599080322861418],[0,0,0,0],[8.999999E+09,8.999999E+09,8.999999E+09,8.999999E+09,8.999999E+09,8.999999E+09]];
    LOCAL CONST Robtarget Tr_meulage_motif_1_246 := [[-62.2027578125,39.22445703125,32.416255859375],[0.368121083594183,-0.372259670766582,0.605815460428718,-0.599080322861418],[0,0,0,0],[8.999999E+09,8.999999E+09,8.999999E+09,8.999999E+09,8.999999E+09,8.999999E+09]];
    LOCAL CONST Robtarget Tr_meulage_motif_1_247 := [[-61.80904296875,39.946640625,31.4991015625],[0.368121083594183,-0.372259670766582,0.605815460428718,-0.599080322861418],[0,0,0,0],[8.999999E+09,8.999999E+09,8.999999E+09,8.999999E+09,8.999999E+09,8.999999E+09]];
    LOCAL CONST Robtarget Tr_meulage_motif_1_248 := [[-61.5239921875,40.4885625,31.076447265625],[0.368121083594183,-0.372259670766582,0.605815460428718,-0.599080322861418],[0,0,0,0],[8.999999E+09,8.999999E+09,8.999999E+09,8.999999E+09,8.999999E+09,8.999999E+09]];
    LOCAL CONST Robtarget Tr_meulage_motif_1_249 := [[-61.005515625,41.49309765625,30.54627734375],[0.368121083594183,-0.372259670766582,0.605815460428718,-0.599080322861418],[0,0,0,0],[8.999999E+09,8.999999E+09,8.999999E+09,8.999999E+09,8.999999E+09,8.999999E+09]];
    LOCAL CONST Robtarget Tr_meulage_motif_1_250 := [[-60.62205078125,42.24616015625,30.282298828125],[0.368121083594183,-0.372259670766582,0.605815460428718,-0.599080322861418],[0,0,0,0],[8.999999E+09,8.999999E+09,8.999999E+09,8.999999E+09,8.999999E+09,8.999999E+09]];
    LOCAL CONST Robtarget Tr_meulage_motif_1_251 := [[-60.20184765625,43.07808203125,30.07790625],[0.368121083594183,-0.372259670766582,0.605815460428718,-0.599080322861418],[0,0,0,0],[8.999999E+09,8.999999E+09,8.999999E+09,8.999999E+09,8.999999E+09,8.999999E+09]];
    LOCAL CONST Robtarget Tr_meulage_motif_1_252 := [[-59.7626484375,43.95590625,29.969388671875],[0.368121083594183,-0.372259670766582,0.605815460428718,-0.599080322861418],[0,0,0,0],[8.999999E+09,8.999999E+09,8.999999E+09,8.999999E+09,8.999999E+09,8.999999E+09]];
    LOCAL CONST Robtarget Tr_meulage_motif_1_253 := [[-59.3185,44.8435546875,29.858810546875],[0.368121083594183,-0.372259670766582,0.605815460428718,-0.599080322861418],[0,0,0,0],[8.999999E+09,8.999999E+09,8.999999E+09,8.999999E+09,8.999999E+09,8.999999E+09]];
    LOCAL CONST Robtarget Tr_meulage_motif_1_254 := [[-58.8745234375,45.73958984375,29.8587734375],[0.368121083594183,-0.372259670766582,0.605815460428718,-0.599080322861418],[0,0,0,0],[8.999999E+09,8.999999E+09,8.999999E+09,8.999999E+09,8.999999E+09,8.999999E+09]];
    LOCAL CONST Robtarget Tr_meulage_motif_1_255 := [[-58.43054296875,46.63562890625,29.858736328125],[0.368121083594183,-0.372259670766582,0.605815460428718,-0.599080322861418],[0,0,0,0],[8.999999E+09,8.999999E+09,8.999999E+09,8.999999E+09,8.999999E+09,8.999999E+09]];
    LOCAL CONST Robtarget Tr_meulage_motif_1_256 := [[-57.98656640625,47.5316640625,29.85869921875],[0.368121083594183,-0.372259670766582,0.605815460428718,-0.599080322861418],[0,0,0,0],[8.999999E+09,8.999999E+09,8.999999E+09,8.999999E+09,8.999999E+09,8.999999E+09]];
    LOCAL CONST Robtarget Tr_meulage_motif_1_257 := [[-57.5425859375,48.427703125,29.858662109375],[0.368121083594183,-0.372259670766582,0.605815460428718,-0.599080322861418],[0,0,0,0],[8.999999E+09,8.999999E+09,8.999999E+09,8.999999E+09,8.999999E+09,8.999999E+09]];
    LOCAL CONST Robtarget Tr_meulage_motif_1_258 := [[-57.09860546875,49.32373828125,29.858625],[0.368121083594183,-0.372259670766582,0.605815460428718,-0.599080322861418],[0,0,0,0],[8.999999E+09,8.999999E+09,8.999999E+09,8.999999E+09,8.999999E+09,8.999999E+09]];
    LOCAL CONST Robtarget Tr_meulage_motif_1_259 := [[-56.65462890625,50.21977734375,29.858587890625],[0.368121083594183,-0.372259670766582,0.605815460428718,-0.599080322861418],[0,0,0,0],[8.999999E+09,8.999999E+09,8.999999E+09,8.999999E+09,8.999999E+09,8.999999E+09]];
    LOCAL CONST Robtarget Tr_meulage_motif_1_260 := [[-56.2106484375,51.1158125,29.85855078125],[0.368121083594183,-0.372259670766582,0.605815460428718,-0.599080322861418],[0,0,0,0],[8.999999E+09,8.999999E+09,8.999999E+09,8.999999E+09,8.999999E+09,8.999999E+09]];
    LOCAL CONST Robtarget Tr_meulage_motif_1_261 := [[-55.766671875,52.0118515625,29.858513671875],[0.368121083594183,-0.372259670766582,0.605815460428718,-0.599080322861418],[0,0,0,0],[8.999999E+09,8.999999E+09,8.999999E+09,8.999999E+09,8.999999E+09,8.999999E+09]];
    LOCAL CONST Robtarget Tr_meulage_motif_1_262 := [[-55.32269140625,52.90788671875,29.8584765625],[0.368121083594183,-0.372259670766582,0.605815460428718,-0.599080322861418],[0,0,0,0],[8.999999E+09,8.999999E+09,8.999999E+09,8.999999E+09,8.999999E+09,8.999999E+09]];
    LOCAL CONST Robtarget Tr_meulage_motif_1_263 := [[-54.8787109375,53.80392578125,29.858439453125],[0.368121083594183,-0.372259670766582,0.605815460428718,-0.599080322861418],[0,0,0,0],[8.999999E+09,8.999999E+09,8.999999E+09,8.999999E+09,8.999999E+09,8.999999E+09]];
    LOCAL CONST Robtarget Tr_meulage_motif_1_264 := [[-54.434734375,54.69996484375,29.85840234375],[0.368121083594183,-0.372259670766582,0.605815460428718,-0.599080322861418],[0,0,0,0],[8.999999E+09,8.999999E+09,8.999999E+09,8.999999E+09,8.999999E+09,8.999999E+09]];
    LOCAL CONST Robtarget Tr_meulage_motif_1_265 := [[-53.99075390625,55.596,29.858365234375],[0.368121083594183,-0.372259670766582,0.605815460428718,-0.599080322861418],[0,0,0,0],[8.999999E+09,8.999999E+09,8.999999E+09,8.999999E+09,8.999999E+09,8.999999E+09]];
    LOCAL CONST Robtarget Tr_meulage_motif_1_266 := [[-53.54677734375,56.4920390625,29.858328125],[0.368121083594183,-0.372259670766582,0.605815460428718,-0.599080322861418],[0,0,0,0],[8.999999E+09,8.999999E+09,8.999999E+09,8.999999E+09,8.999999E+09,8.999999E+09]];
    LOCAL CONST Robtarget Tr_meulage_motif_1_267 := [[-53.102796875,57.38807421875,29.858291015625],[0.368121083594183,-0.372259670766582,0.605815460428718,-0.599080322861418],[0,0,0,0],[8.999999E+09,8.999999E+09,8.999999E+09,8.999999E+09,8.999999E+09,8.999999E+09]];
    LOCAL CONST Robtarget Tr_meulage_motif_1_268 := [[-52.65881640625,58.28411328125,29.85825390625],[0.368121083594183,-0.372259670766582,0.605815460428718,-0.599080322861418],[0,0,0,0],[8.999999E+09,8.999999E+09,8.999999E+09,8.999999E+09,8.999999E+09,8.999999E+09]];
    LOCAL CONST Robtarget Tr_meulage_motif_1_269 := [[-52.21483984375,59.1801484375,29.858216796875],[0.368121083594183,-0.372259670766582,0.605815460428718,-0.599080322861418],[0,0,0,0],[8.999999E+09,8.999999E+09,8.999999E+09,8.999999E+09,8.999999E+09,8.999999E+09]];
    LOCAL CONST Robtarget Tr_meulage_motif_1_270 := [[-51.770859375,60.0761875,29.8581796875],[0.368121083594183,-0.372259670766582,0.605815460428718,-0.599080322861418],[0,0,0,0],[8.999999E+09,8.999999E+09,8.999999E+09,8.999999E+09,8.999999E+09,8.999999E+09]];
    LOCAL CONST Robtarget Tr_meulage_motif_1_271 := [[-51.32687890625,60.97222265625,29.858140625],[0.368121083594183,-0.372259670766582,0.605815460428718,-0.599080322861418],[0,0,0,0],[8.999999E+09,8.999999E+09,8.999999E+09,8.999999E+09,8.999999E+09,8.999999E+09]];
    LOCAL CONST Robtarget Tr_meulage_motif_1_272 := [[-50.88290234375,61.86826171875,29.858103515625],[0.368121083594183,-0.372259670766582,0.605815460428718,-0.599080322861418],[0,0,0,0],[8.999999E+09,8.999999E+09,8.999999E+09,8.999999E+09,8.999999E+09,8.999999E+09]];
    LOCAL CONST Robtarget Tr_meulage_motif_1_273 := [[-50.438921875,62.764296875,29.85806640625],[0.368121083594183,-0.372259670766582,0.605815460428718,-0.599080322861418],[0,0,0,0],[8.999999E+09,8.999999E+09,8.999999E+09,8.999999E+09,8.999999E+09,8.999999E+09]];
    LOCAL CONST Robtarget Tr_meulage_motif_1_274 := [[-49.9949453125,63.6603359375,29.858029296875],[0.368121083594183,-0.372259670766582,0.605815460428718,-0.599080322861418],[0,0,0,0],[8.999999E+09,8.999999E+09,8.999999E+09,8.999999E+09,8.999999E+09,8.999999E+09]];
    LOCAL CONST Robtarget Tr_meulage_motif_1_275 := [[-49.55096484375,64.55637109375,29.8579921875],[0.368121083594183,-0.372259670766582,0.605815460428718,-0.599080322861418],[0,0,0,0],[8.999999E+09,8.999999E+09,8.999999E+09,8.999999E+09,8.999999E+09,8.999999E+09]];
    LOCAL CONST Robtarget Tr_meulage_motif_1_276 := [[-49.106984375,65.45241015625,29.857955078125],[0.368121083594183,-0.372259670766582,0.605815460428718,-0.599080322861418],[0,0,0,0],[8.999999E+09,8.999999E+09,8.999999E+09,8.999999E+09,8.999999E+09,8.999999E+09]];
    LOCAL CONST Robtarget Tr_meulage_motif_1_277 := [[-48.6630078125,66.3484453125,29.85791796875],[0.368121083594183,-0.372259670766582,0.605815460428718,-0.599080322861418],[0,0,0,0],[8.999999E+09,8.999999E+09,8.999999E+09,8.999999E+09,8.999999E+09,8.999999E+09]];
    LOCAL CONST Robtarget Tr_meulage_motif_1_278 := [[-48.21902734375,67.244484375,29.857880859375],[0.368121083594183,-0.372259670766582,0.605815460428718,-0.599080322861418],[0,0,0,0],[8.999999E+09,8.999999E+09,8.999999E+09,8.999999E+09,8.999999E+09,8.999999E+09]];
    LOCAL CONST Robtarget Tr_meulage_motif_1_279 := [[-47.77505078125,68.1405234375,29.85784375],[0.368121083594183,-0.372259670766582,0.605815460428718,-0.599080322861418],[0,0,0,0],[8.999999E+09,8.999999E+09,8.999999E+09,8.999999E+09,8.999999E+09,8.999999E+09]];
    LOCAL CONST Robtarget Tr_meulage_motif_1_280 := [[-47.3310703125,69.0365546875,29.857806640625],[0.368121083594183,-0.372259670766582,0.605815460428718,-0.599080322861418],[0,0,0,0],[8.999999E+09,8.999999E+09,8.999999E+09,8.999999E+09,8.999999E+09,8.999999E+09]];
    LOCAL CONST Robtarget Tr_meulage_motif_1_281 := [[-46.88708984375,69.93259375,29.85776953125],[0.368121083594183,-0.372259670766582,0.605815460428718,-0.599080322861418],[0,0,0,0],[8.999999E+09,8.999999E+09,8.999999E+09,8.999999E+09,8.999999E+09,8.999999E+09]];
    LOCAL CONST Robtarget Tr_meulage_motif_1_282 := [[-46.44311328125,70.8286328125,29.857732421875],[0.368121083594183,-0.372259670766582,0.605815460428718,-0.599080322861418],[0,0,0,0],[8.999999E+09,8.999999E+09,8.999999E+09,8.999999E+09,8.999999E+09,8.999999E+09]];
    LOCAL CONST Robtarget Tr_meulage_motif_1_283 := [[-45.9991328125,71.724671875,29.8576953125],[0.368121083594183,-0.372259670766582,0.605815460428718,-0.599080322861418],[0,0,0,0],[8.999999E+09,8.999999E+09,8.999999E+09,8.999999E+09,8.999999E+09,8.999999E+09]];
    LOCAL CONST Robtarget Tr_meulage_motif_1_284 := [[-45.55515625,72.6207109375,29.857658203125],[0.368121083594183,-0.372259670766582,0.605815460428718,-0.599080322861418],[0,0,0,0],[8.999999E+09,8.999999E+09,8.999999E+09,8.999999E+09,8.999999E+09,8.999999E+09]];
    LOCAL CONST Robtarget Tr_meulage_motif_1_285 := [[-45.11117578125,73.5167421875,29.85762109375],[0.368121083594183,-0.372259670766582,0.605815460428718,-0.599080322861418],[0,0,0,0],[8.999999E+09,8.999999E+09,8.999999E+09,8.999999E+09,8.999999E+09,8.999999E+09]];
    LOCAL CONST Robtarget Tr_meulage_motif_1_286 := [[-44.6671953125,74.41278125,29.857583984375],[0.368121083594183,-0.372259670766582,0.605815460428718,-0.599080322861418],[0,0,0,0],[8.999999E+09,8.999999E+09,8.999999E+09,8.999999E+09,8.999999E+09,8.999999E+09]];
    LOCAL CONST Robtarget Tr_meulage_motif_1_287 := [[-44.22321875,75.3088203125,29.857546875],[0.368121083594183,-0.372259670766582,0.605815460428718,-0.599080322861418],[0,0,0,0],[8.999999E+09,8.999999E+09,8.999999E+09,8.999999E+09,8.999999E+09,8.999999E+09]];
    LOCAL CONST Robtarget Tr_meulage_motif_1_288 := [[-43.77923828125,76.204859375,29.857509765625],[0.368121083594183,-0.372259670766582,0.605815460428718,-0.599080322861418],[0,0,0,0],[8.999999E+09,8.999999E+09,8.999999E+09,8.999999E+09,8.999999E+09,8.999999E+09]];
    LOCAL CONST Robtarget Tr_meulage_motif_1_289 := [[-43.33526171875,77.100890625,29.85747265625],[0.368121083594183,-0.372259670766582,0.605815460428718,-0.599080322861418],[0,0,0,0],[8.999999E+09,8.999999E+09,8.999999E+09,8.999999E+09,8.999999E+09,8.999999E+09]];
    LOCAL CONST Robtarget Tr_meulage_motif_1_290 := [[-42.89128125,77.9969296875,29.857435546875],[0.368121083594183,-0.372259670766582,0.605815460428718,-0.599080322861418],[0,0,0,0],[8.999999E+09,8.999999E+09,8.999999E+09,8.999999E+09,8.999999E+09,8.999999E+09]];
    LOCAL CONST Robtarget Tr_meulage_motif_1_291 := [[-42.44730078125,78.89296875,29.8573984375],[0.368121083594183,-0.372259670766582,0.605815460428718,-0.599080322861418],[0,0,0,0],[8.999999E+09,8.999999E+09,8.999999E+09,8.999999E+09,8.999999E+09,8.999999E+09]];
    LOCAL CONST Robtarget Tr_meulage_motif_1_292 := [[-42.00332421875,79.7890078125,29.857361328125],[0.368121083594183,-0.372259670766582,0.605815460428718,-0.599080322861418],[0,0,0,0],[8.999999E+09,8.999999E+09,8.999999E+09,8.999999E+09,8.999999E+09,8.999999E+09]];
    LOCAL CONST Robtarget Tr_meulage_motif_1_293 := [[-41.55934375,80.6850390625,29.85732421875],[0.368121083594183,-0.372259670766582,0.605815460428718,-0.599080322861418],[0,0,0,0],[8.999999E+09,8.999999E+09,8.999999E+09,8.999999E+09,8.999999E+09,8.999999E+09]];
    LOCAL CONST Robtarget Tr_meulage_motif_1_294 := [[-41.11536328125,81.581078125,29.857287109375],[0.368121083594183,-0.372259670766582,0.605815460428718,-0.599080322861418],[0,0,0,0],[8.999999E+09,8.999999E+09,8.999999E+09,8.999999E+09,8.999999E+09,8.999999E+09]];

